KUKA KRL program: EPS_2_251806_MH46A_A_20260212042242.src

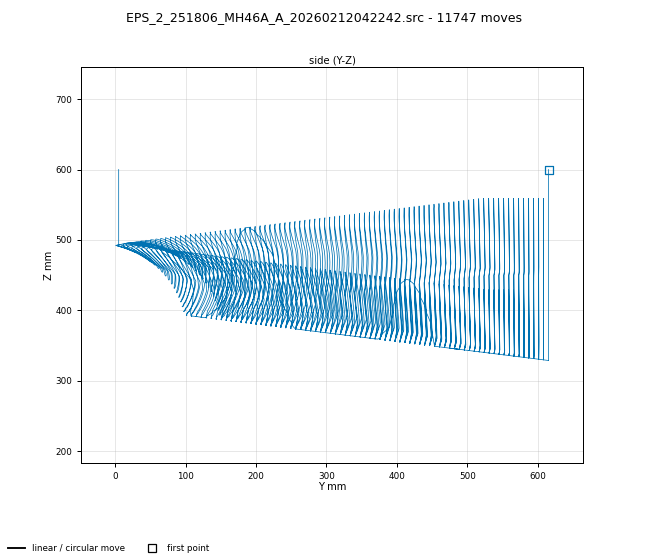
[picture p0: tool path of EPS_2_251806_MH46A_A_20260212042242.src, 11747 of 11749 moves have a stored position in this frame; points joined in program order, loops and branches not executed]
&ACCESS RVP
&REL 4
&COMMENT QRS 19112012
&PARAM EDITMASK = *
DEF PART()
EXT BAS (BAS_COMMAND :IN,REAL :IN )
INT I
BAS (#INITMOV,0 )

;KUKA QRS Post kuka4.cps  Date:22-06-2017 !

File_ID=3018

QRS_PRE_INIT()

;Init var - Until changes are made in qrs_pre_init
Outlet_Square_prg=0
Inlet_1_Square_prg=0
Inlet_2_Square_prg=0
Inlet_3_Square_prg=0
Inlet_4_Square_prg=0
Inlet_5_Square_prg=0

Outlet_1={X 0.000, Y 520.860, Z 458.500, B 0.000, E1 0.000 }
Inlet_1={X 0.000, Y 530.280, Z 328.500, B 0.000, E1 188.000 }
Outlet_1_type=201
Inlet_1_type=201
;QRS#1=Sidecore dimensions
;QRS#2=200-8" PVC SDR 35
;QRS#3=200-8" PVC SDR 35
;QRS#4=
;QRS#5=
;QRS#6=
;QRS#7=
;QRS#8=
;QRS#9=12-08 PSX
;QRS#10=12-08 PSX
;QRS#11=
;QRS#12=
;QRS#13=
;QRS#14=
;QRS#15=
;QRS#16=1220x127x838 2,75'
;QRS#17=EPS Height
;QRS#18=559
;QRS#19=*
;QRS#20= UPDATED VERSION 22-06-2017
;QRS#21=*
Outlet_Square=0100
Inlet_1_Square=0100
Inlet_2_Square=0
Inlet_3_Square=0
Inlet_4_Square=0
Inlet_5_Square=0
Mill_Square=1
Outlet_Square_Prg=204
Inlet_1_Square_prg=204

QRS_INIT()

$ADVANCE=5

; T1
PTP {E1 173.606,E2 173.606}
PTP {X 0,Y 615.511,A -85,B 0,C 180,E1 173.606,E2 173.606,E3 0,E4 0,E5 0,E6 0}
QRS_SPEED_INIT()
LIN {X 0,Y 615.511,Z 600,A -85,B 0,C 180,E1 173.606,E2 173.606,E3 0,E4 0,E5 0,E6 0} C_VEL
LIN {X 0,Y 615.511,Z 338.873,A -85,B 0,C 180,E1 173.606,E2 173.606} C_VEL
LIN {X 0,Y 615.511,Z 330.7,A -85,B 0,C 180,E1 173.606,E2 173.606} C_VEL
LIN {X 0,Y 615.495,Z 328.7,A -85,B 0,C 180,E1 173.42,E2 173.42} C_VEL
LIN {X 0,Y 615.496,Z 328.696,A -85,B 0,C 180,E1 170.801,E2 170.801} C_VEL
LIN {X 0,Y 615.477,Z 328.699,A -85,B 0,C 180,E1 168.139,E2 168.139} C_VEL
LIN {X 0,Y 615.495,Z 328.7,A -85,B 0,C 180,E1 165.451,E2 165.451} C_VEL
LIN {X 0,Y 615.495,Z 328.694,A -85,B 0,C 180,E1 162.729,E2 162.729} C_VEL
LIN {X 0,Y 615.493,Z 328.701,A -85,B 0,C 180,E1 159.967,E2 159.967} C_VEL
LIN {X 0,Y 615.487,Z 328.696,A -85,B 0,C 180,E1 157.155,E2 157.155} C_VEL
LIN {X 0,Y 615.499,Z 328.7,A -85,B 0,C 180,E1 154.284,E2 154.284} C_VEL
LIN {X 0,Y 615.478,Z 328.698,A -85,B 0,C 180,E1 151.552,E2 151.552} C_VEL
LIN {X 0,Y 615.492,Z 328.698,A -85,B 0,C 180,E1 148.914,E2 148.914} C_VEL
LIN {X 0,Y 615.498,Z 328.7,A -85,B 0,C 180,E1 146.465,E2 146.465} C_VEL
LIN {X 0,Y 615.494,Z 328.7,A -85,B 0,C 180,E1 144.166,E2 144.166} C_VEL
LIN {X 0,Y 615.491,Z 328.701,A -85,B 0,C 180,E1 141.931,E2 141.931} C_VEL
LIN {X 0,Y 615.491,Z 328.696,A -85,B 0,C 180,E1 139.393,E2 139.393} C_VEL
LIN {X 0,Y 615.482,Z 328.698,A -85,B 0,C 180,E1 136.754,E2 136.754} C_VEL
LIN {X 0,Y 615.491,Z 328.699,A -85,B 0,C 180,E1 133.997,E2 133.997} C_VEL
LIN {X 0,Y 615.493,Z 328.696,A -85,B 0,C 180,E1 131.094,E2 131.094} C_VEL
LIN {X 0,Y 615.484,Z 328.698,A -85,B 0,C 180,E1 128.905,E2 128.905} C_VEL
LIN {X 0,Y 615.49,Z 328.699,A -85,B 0,C 180,E1 126.425,E2 126.425} C_VEL
LIN {X 0,Y 615.496,Z 328.694,A -85,B 0,C 180,E1 123.534,E2 123.534} C_VEL
LIN {X 0,Y 615.487,Z 328.698,A -85,B 0,C 180,E1 120.92,E2 120.92} C_VEL
LIN {X 0,Y 615.498,Z 328.7,A -85,B 0,C 180,E1 118.451,E2 118.451} C_VEL
LIN {X 0,Y 615.499,Z 328.694,A -85,B 0,C 180,E1 115.57,E2 115.57} C_VEL
LIN {X 0,Y 615.492,Z 328.701,A -85,B 0,C 180,E1 112.845,E2 112.845} C_VEL
LIN {X 0,Y 615.482,Z 328.697,A -85,B 0,C 180,E1 110.033,E2 110.033} C_VEL
LIN {X 0,Y 615.495,Z 328.7,A -85,B 0,C 180,E1 107.271,E2 107.271} C_VEL
LIN {X 0,Y 615.484,Z 328.697,A -85,B 0,C 180,E1 104.55,E2 104.55} C_VEL
LIN {X 0,Y 615.49,Z 328.697,A -85,B 0,C 180,E1 101.861,E2 101.861} C_VEL
LIN {X 0,Y 615.495,Z 328.698,A -85,B 0,C 180,E1 99.199,E2 99.199} C_VEL
LIN {X 0,Y 615.479,Z 328.698,A -85,B 0,C 180,E1 96.557,E2 96.557} C_VEL
LIN {X 0,Y 615.488,Z 328.7,A -85,B 0,C 180,E1 93.601,E2 93.601} C_VEL
LIN {X 0,Y 615.482,Z 328.699,A -85,B 0,C 180,E1 93.478,E2 93.478} C_VEL
LIN {X 0,Y 615.482,Z 341.691,A -85,B 0,C 180,E1 93.151,E2 93.151} C_VEL
LIN {X 0,Y 615.495,Z 354.109,A -85,B 0,C 180,E1 92.7,E2 92.7} C_VEL
LIN {X 0,Y 615.492,Z 366.017,A -85,B 0,C 180,E1 92.127,E2 92.127} C_VEL
LIN {X 0,Y 615.495,Z 376.719,A -85,B 0,C 180,E1 91.473,E2 91.473} C_VEL
LIN {X 0,Y 615.498,Z 387.355,A -85,B 0,C 180,E1 90.655,E2 90.655} C_VEL
LIN {X 0,Y 615.499,Z 396.028,A -85,B 0,C 180,E1 89.837,E2 89.837} C_VEL
LIN {X 0,Y 615.496,Z 404.503,A -85,B 0,C 180,E1 88.856,E2 88.856} C_VEL
LIN {X 0,Y 615.496,Z 411.299,A -85,B 0,C 180,E1 87.874,E2 87.874} C_VEL
LIN {X 0,Y 615.497,Z 417.556,A -85,B 0,C 180,E1 86.728,E2 86.728} C_VEL
LIN {X 0,Y 615.495,Z 421.662,A -85,B 0,C 180,E1 85.744,E2 85.744} C_VEL
LIN {X 0,Y 615.495,Z 424.735,A -85,B 0,C 180,E1 84.759,E2 84.759} C_VEL
LIN {X 0,Y 615.499,Z 426.265,A -85,B 0,C 180,E1 84.102,E2 84.102} C_VEL
LIN {X 0,Y 615.496,Z 427.396,A -85,B 0,C 180,E1 83.42,E2 83.42} C_VEL
LIN {X 0,Y 615.497,Z 428.353,A -85,B 0,C 180,E1 82.125,E2 82.125} C_VEL
LIN {X 0,Y 615.494,Z 428.277,A -85,B 0,C 180,E1 81.464,E2 81.464} C_VEL
LIN {X 0,Y 615.497,Z 427.763,A -85,B 0,C 180,E1 80.802,E2 80.802} C_VEL
LIN {X 0,Y 615.499,Z 426.851,A -85,B 0,C 180,E1 80.138,E2 80.138} C_VEL
LIN {X 0,Y 615.494,Z 424.63,A -85,B 0,C 180,E1 79.112,E2 79.112} C_VEL
LIN {X 0,Y 615.494,Z 421.565,A -85,B 0,C 180,E1 78.14,E2 78.14} C_VEL
LIN {X 0,Y 615.498,Z 417.326,A -85,B 0,C 180,E1 77.135,E2 77.135} C_VEL
LIN {X 0,Y 615.497,Z 411.481,A -85,B 0,C 180,E1 76.066,E2 76.066} C_VEL
LIN {X 0,Y 615.496,Z 404.943,A -85,B 0,C 180,E1 75.113,E2 75.113} C_VEL
LIN {X 0,Y 615.499,Z 397.842,A -85,B 0,C 180,E1 74.266,E2 74.266} C_VEL
LIN {X 0,Y 615.497,Z 389.207,A -85,B 0,C 180,E1 73.414,E2 73.414} C_VEL
LIN {X 0,Y 615.498,Z 378.423,A -85,B 0,C 180,E1 72.559,E2 72.559} C_VEL
LIN {X 0,Y 615.482,Z 367.809,A -85,B 0,C 180,E1 71.881,E2 71.881} C_VEL
LIN {X 0,Y 615.493,Z 357.48,A -85,B 0,C 180,E1 71.355,E2 71.355} C_VEL
LIN {X 0,Y 615.48,Z 345.396,A -85,B 0,C 180,E1 70.879,E2 70.879} C_VEL
LIN {X 0,Y 615.491,Z 333.153,A -85,B 0,C 180,E1 70.533,E2 70.533} C_VEL
LIN {X 0,Y 615.492,Z 328.702,A -85,B 0,C 180,E1 70.424,E2 70.424} C_VEL
LIN {X 0,Y 615.483,Z 328.7,A -85,B 0,C 180,E1 67.656,E2 67.656} C_VEL
LIN {X 0,Y 615.479,Z 328.7,A -85,B 0,C 180,E1 65.008,E2 65.008} C_VEL
LIN {X 0,Y 615.476,Z 328.701,A -85,B 0,C 180,E1 62.823,E2 62.823} C_VEL
LIN {X 0,Y 615.482,Z 328.7,A -85,B 0,C 180,E1 60.207,E2 60.207} C_VEL
LIN {X 0,Y 615.494,Z 328.7,A -85,B 0,C 180,E1 57.543,E2 57.543} C_VEL
LIN {X 0,Y 615.484,Z 328.699,A -85,B 0,C 180,E1 55.185,E2 55.185} C_VEL
LIN {X 0,Y 615.488,Z 328.699,A -85,B 0,C 180,E1 52.759,E2 52.759} C_VEL
LIN {X 0,Y 615.482,Z 328.699,A -85,B 0,C 180,E1 49.912,E2 49.912} C_VEL
LIN {X 0,Y 615.499,Z 328.698,A -85,B 0,C 180,E1 47.649,E2 47.649} C_VEL
LIN {X 0,Y 615.486,Z 328.698,A -85,B 0,C 180,E1 44.932,E2 44.932} C_VEL
LIN {X 0,Y 615.485,Z 328.698,A -85,B 0,C 180,E1 42.081,E2 42.081} C_VEL
LIN {X 0,Y 615.497,Z 328.697,A -85,B 0,C 180,E1 39.75,E2 39.75} C_VEL
LIN {X 0,Y 615.492,Z 328.697,A -85,B 0,C 180,E1 36.938,E2 36.938} C_VEL
LIN {X 0,Y 615.497,Z 328.698,A -85,B 0,C 180,E1 34.703,E2 34.703} C_VEL
LIN {X 0,Y 615.482,Z 328.7,A -85,B 0,C 180,E1 32.331,E2 32.331} C_VEL
LIN {X 0,Y 615.496,Z 328.697,A -85,B 0,C 180,E1 29.797,E2 29.797} C_VEL
LIN {X 0,Y 615.499,Z 328.695,A -85,B 0,C 180,E1 27.048,E2 27.048} C_VEL
LIN {X 0,Y 615.492,Z 328.697,A -85,B 0,C 180,E1 24.272,E2 24.272} C_VEL
LIN {X 0,Y 615.495,Z 328.698,A -85,B 0,C 180,E1 21.432,E2 21.432} C_VEL
LIN {X 0,Y 615.495,Z 328.701,A -85,B 0,C 180,E1 18.608,E2 18.608} C_VEL
LIN {X 0,Y 615.489,Z 328.698,A -85,B 0,C 180,E1 15.905,E2 15.905} C_VEL
LIN {X 0,Y 615.496,Z 328.696,A -85,B 0,C 180,E1 13.201,E2 13.201} C_VEL
LIN {X 0,Y 615.495,Z 328.699,A -85,B 0,C 180,E1 10.527,E2 10.527} C_VEL
LIN {X 0,Y 615.485,Z 328.7,A -85,B 0,C 180,E1 7.876,E2 7.876} C_VEL
LIN {X 0,Y 615.491,Z 328.697,A -85,B 0,C 180,E1 5.241,E2 5.241} C_VEL
LIN {X 0,Y 615.496,Z 328.7,A -85,B 0,C 180,E1 2.618,E2 2.618} C_VEL
LIN {X 0,Y 615.484,Z 328.699,A -85,B 0,C 180,E1 0,E2 0} C_VEL
LIN {X 0,Y 615.49,Z 328.698,A -85,B 0,C 180,E1 -2.618,E2 -2.618} C_VEL
LIN {X 0,Y 615.497,Z 328.7,A -85,B 0,C 180,E1 -5.241,E2 -5.241} C_VEL
LIN {X 0,Y 615.479,Z 328.7,A -85,B 0,C 180,E1 -7.876,E2 -7.876} C_VEL
LIN {X 0,Y 615.487,Z 328.699,A -85,B 0,C 180,E1 -10.527,E2 -10.527} C_VEL
LIN {X 0,Y 615.496,Z 328.7,A -85,B 0,C 180,E1 -13.201,E2 -13.201} C_VEL
LIN {X 0,Y 615.477,Z 328.701,A -85,B 0,C 180,E1 -15.905,E2 -15.905} C_VEL
LIN {X 0,Y 615.479,Z 328.7,A -85,B 0,C 180,E1 -18.646,E2 -18.646} C_VEL
LIN {X 0,Y 615.485,Z 328.7,A -85,B 0,C 180,E1 -21.432,E2 -21.432} C_VEL
LIN {X 0,Y 615.489,Z 328.701,A -85,B 0,C 180,E1 -24.272,E2 -24.272} C_VEL
LIN {X 0,Y 615.493,Z 328.701,A -85,B 0,C 180,E1 -27.177,E2 -27.177} C_VEL
LIN {X 0,Y 615.499,Z 328.7,A -85,B 0,C 180,E1 -30.159,E2 -30.159} C_VEL
LIN {X 0,Y 615.485,Z 328.699,A -85,B 0,C 180,E1 -32.458,E2 -32.458} C_VEL
LIN {X 0,Y 615.491,Z 328.697,A -85,B 0,C 180,E1 -34.815,E2 -34.815} C_VEL
LIN {X 0,Y 615.495,Z 328.699,A -85,B 0,C 180,E1 -37.242,E2 -37.242} C_VEL
LIN {X 0,Y 615.498,Z 328.7,A -85,B 0,C 180,E1 -40.091,E2 -40.091} C_VEL
LIN {X 0,Y 615.492,Z 328.7,A -85,B 0,C 180,E1 -43.049,E2 -43.049} C_VEL
LIN {X 0,Y 615.49,Z 328.7,A -85,B 0,C 180,E1 -46.002,E2 -46.002} C_VEL
LIN {X 0,Y 615.496,Z 328.698,A -85,B 0,C 180,E1 -48.905,E2 -48.905} C_VEL
LIN {X 0,Y 615.497,Z 328.701,A -85,B 0,C 180,E1 -51.097,E2 -51.097} C_VEL
LIN {X 0,Y 615.492,Z 328.697,A -85,B 0,C 180,E1 -53.576,E2 -53.576} C_VEL
LIN {X 0,Y 615.489,Z 328.805,A -85,B 0,C 180,E1 -54.611,E2 -54.611} C_VEL
LIN {X 0,Y 615.491,Z 341.278,A -85,B 0,C 180,E1 -57.155,E2 -57.155} C_VEL
LIN {X 0,Y 615.495,Z 354.171,A -85,B 0,C 180,E1 -59.841,E2 -59.841} C_VEL
LIN {X 0,Y 615.495,Z 366.88,A -85,B 0,C 180,E1 -62.455,E2 -62.455} C_VEL
LIN {X 0,Y 615.478,Z 379.58,A -85,B 0,C 180,E1 -65.008,E2 -65.008} C_VEL
LIN {X 0,Y 615.484,Z 394.081,A -85,B 0,C 180,E1 -67.864,E2 -67.864} C_VEL
LIN {X 0,Y 615.485,Z 408.57,A -85,B 0,C 180,E1 -70.663,E2 -70.663} C_VEL
LIN {X 0,Y 615.496,Z 423.857,A -85,B 0,C 180,E1 -73.567,E2 -73.567} C_VEL
LIN {X 0,Y 615.493,Z 439.318,A -85,B 0,C 180,E1 -76.463,E2 -76.463} C_VEL
LIN {X 0,Y 615.49,Z 449.367,A -85,B 0,C 180,E1 -78.328,E2 -78.328} C_VEL
LIN {X 0,Y 615.478,Z 464.088,A -85,B 0,C 180,E1 -78.599,E2 -78.599} C_VEL
LIN {X 0,Y 615.481,Z 476.501,A -85,B 0,C 180,E1 -78.96,E2 -78.96} C_VEL
LIN {X 0,Y 615.481,Z 489.034,A -85,B 0,C 180,E1 -79.473,E2 -79.473} C_VEL
LIN {X 0,Y 615.491,Z 499.989,A -85,B 0,C 180,E1 -80.055,E2 -80.055} C_VEL
LIN {X 0,Y 615.499,Z 511.174,A -85,B 0,C 180,E1 -80.802,E2 -80.802} C_VEL
LIN {X 0,Y 615.498,Z 521.05,A -85,B 0,C 180,E1 -81.629,E2 -81.629} C_VEL
LIN {X 0,Y 615.498,Z 530.61,A -85,B 0,C 180,E1 -82.62,E2 -82.62} C_VEL
LIN {X 0,Y 615.496,Z 538.206,A -85,B 0,C 180,E1 -83.609,E2 -83.609} C_VEL
LIN {X 0,Y 615.498,Z 545.207,A -85,B 0,C 180,E1 -84.759,E2 -84.759} C_VEL
LIN {X 0,Y 615.493,Z 549.854,A -85,B 0,C 180,E1 -85.744,E2 -85.744} C_VEL
LIN {X 0,Y 615.495,Z 553.4,A -85,B 0,C 180,E1 -86.728,E2 -86.728} C_VEL
LIN {X 0,Y 615.497,Z 555.234,A -85,B 0,C 180,E1 -87.383,E2 -87.383} C_VEL
LIN {X 0,Y 615.499,Z 556.608,A -85,B 0,C 180,E1 -88.037,E2 -88.037} C_VEL
LIN {X 0,Y 615.496,Z 558.174,A -85,B 0,C 180,E1 -89.346,E2 -89.346} C_VEL
LIN {X 0,Y 615.494,Z 558.389,A -85,B 0,C 180,E1 -90,E2 -90} C_VEL
LIN {X 0,Y 615.496,Z 557.579,A -85,B 0,C 180,E1 -91.309,E2 -91.309} C_VEL
LIN {X 0,Y 615.499,Z 556.607,A -85,B 0,C 180,E1 -91.964,E2 -91.964} C_VEL
LIN {X 0,Y 615.497,Z 555.232,A -85,B 0,C 180,E1 -92.618,E2 -92.618} C_VEL
LIN {X 0,Y 615.496,Z 552.348,A -85,B 0,C 180,E1 -93.601,E2 -93.601} C_VEL
LIN {X 0,Y 615.498,Z 548.439,A -85,B 0,C 180,E1 -94.585,E2 -94.585} C_VEL
LIN {X 0,Y 615.499,Z 543.402,A -85,B 0,C 180,E1 -95.57,E2 -95.57} C_VEL
LIN {X 0,Y 615.497,Z 536.869,A -85,B 0,C 180,E1 -96.583,E2 -96.583} C_VEL
LIN {X 0,Y 615.497,Z 529.129,A -85,B 0,C 180,E1 -97.546,E2 -97.546} C_VEL
LIN {X 0,Y 615.498,Z 521.04,A -85,B 0,C 180,E1 -98.372,E2 -98.372} C_VEL
LIN {X 0,Y 615.499,Z 511.161,A -85,B 0,C 180,E1 -99.199,E2 -99.199} C_VEL
LIN {X 0,Y 615.491,Z 499.973,A -85,B 0,C 180,E1 -99.946,E2 -99.946} C_VEL
LIN {X 0,Y 615.481,Z 489.013,A -85,B 0,C 180,E1 -100.527,E2 -100.527} C_VEL
LIN {X 0,Y 615.484,Z 476.479,A -85,B 0,C 180,E1 -101.04,E2 -101.04} C_VEL
LIN {X 0,Y 615.478,Z 464.046,A -85,B 0,C 180,E1 -101.402,E2 -101.402} C_VEL
LIN {X 0,Y 615.49,Z 449.249,A -85,B 0,C 180,E1 -101.694,E2 -101.694} C_VEL
LIN {X 0,Y 615.483,Z 433.893,A -85,B 0,C 180,E1 -104.55,E2 -104.55} C_VEL
LIN {X 0,Y 615.478,Z 419.426,A -85,B 0,C 180,E1 -107.271,E2 -107.271} C_VEL
LIN {X 0,Y 615.479,Z 404.947,A -85,B 0,C 180,E1 -110.034,E2 -110.034} C_VEL
LIN {X 0,Y 615.492,Z 390.453,A -85,B 0,C 180,E1 -112.845,E2 -112.845} C_VEL
LIN {X 0,Y 615.492,Z 375.947,A -85,B 0,C 180,E1 -115.716,E2 -115.716} C_VEL
LIN {X 0,Y 615.491,Z 362.442,A -85,B 0,C 180,E1 -118.451,E2 -118.451} C_VEL
LIN {X 0,Y 615.485,Z 349.75,A -85,B 0,C 180,E1 -121.085,E2 -121.085} C_VEL
LIN {X 0,Y 615.495,Z 337.872,A -85,B 0,C 180,E1 -123.535,E2 -123.535} C_VEL
LIN {X 0,Y 615.488,Z 328.696,A -85,B 0,C 180,E1 -125.466,E2 -125.466} C_VEL
LIN {X 0,Y 615.483,Z 328.7,A -85,B 0,C 180,E1 -128.069,E2 -128.069} C_VEL
LIN {X 0,Y 615.492,Z 328.7,A -85,B 0,C 180,E1 -130.607,E2 -130.607} C_VEL
LIN {X 0,Y 615.497,Z 328.694,A -85,B 0,C 180,E1 -133.244,E2 -133.244} C_VEL
LIN {X 0,Y 615.484,Z 328.701,A -85,B 0,C 180,E1 -136.004,E2 -136.004} C_VEL
LIN {X 0,Y 615.483,Z 328.697,A -85,B 0,C 180,E1 -138.907,E2 -138.907} C_VEL
LIN {X 0,Y 615.493,Z 328.695,A -85,B 0,C 180,E1 -141.096,E2 -141.096} C_VEL
LIN {X 0,Y 615.478,Z 328.699,A -85,B 0,C 180,E1 -143.574,E2 -143.574} C_VEL
LIN {X 0,Y 615.489,Z 328.698,A -85,B 0,C 180,E1 -145.978,E2 -145.978} C_VEL
LIN {X 0,Y 615.495,Z 328.698,A -85,B 0,C 180,E1 -148.315,E2 -148.315} C_VEL
LIN {X 0,Y 615.49,Z 328.699,A -85,B 0,C 180,E1 -150.594,E2 -150.594} C_VEL
LIN {X 0,Y 615.497,Z 328.7,A -85,B 0,C 180,E1 -152.954,E2 -152.954} C_VEL
LIN {X 0,Y 615.492,Z 328.695,A -85,B 0,C 180,E1 -155.728,E2 -155.728} C_VEL
LIN {X 0,Y 615.498,Z 328.7,A -85,B 0,C 180,E1 -158.569,E2 -158.569} C_VEL
LIN {X 0,Y 615.477,Z 328.699,A -85,B 0,C 180,E1 -161.4,E2 -161.4} C_VEL
LIN {X 0,Y 615.494,Z 328.699,A -85,B 0,C 180,E1 -164.095,E2 -164.095} C_VEL
LIN {X 0,Y 615.494,Z 328.696,A -85,B 0,C 180,E1 -166.799,E2 -166.799} C_VEL
LIN {X 0,Y 615.486,Z 328.698,A -85,B 0,C 180,E1 -169.473,E2 -169.473} C_VEL
LIN {X 0,Y 615.492,Z 328.7,A -85,B 0,C 180,E1 -172.125,E2 -172.125} C_VEL
LIN {X 0,Y 615.488,Z 328.696,A -85,B 0,C 180,E1 -174.759,E2 -174.759} C_VEL
LIN {X 0,Y 615.488,Z 328.698,A -85,B 0,C 180,E1 -177.382,E2 -177.382} C_VEL
LIN {X 0,Y 615.492,Z 328.7,A -85,B 0,C 180,E1 -180,E2 -180} C_VEL
LIN {X 0,Y 615.489,Z 328.696,A -85,B 0,C 180,E1 -182.618,E2 -182.618} C_VEL
LIN {X 0,Y 615.487,Z 328.698,A -85,B 0,C 180,E1 -185.241,E2 -185.241} C_VEL
LIN {X 0,Y 615.495,Z 328.7,A -85,B 0,C 180,E1 -186.58,E2 -186.58} C_VEL
LIN {X 0,Y 614.816,Z 328.843,A -85,B 0,C 180,E1 -187.126,E2 -187.126} C_VEL
LIN {X 0,Y 611.983,Z 329.256,A -85,B 0,C 180,E1 -188.012,E2 -188.012} C_VEL
LIN {X 0,Y 609.593,Z 329.565,A -85,B 0,C 180,E1 -188.724,E2 -188.724} C_VEL
LIN {X 0,Y 608.558,Z 329.683,A -85,B 0,C 180,E1 -189.274,E2 -189.274} C_VEL
LIN {X 0,Y 608.468,Z 329.693,A -85,B 0,C 180,E1 -189.46,E2 -189.46} C_VEL
LIN {X 0,Y 608.456,Z 329.696,A -85,B 0,C 180,E1 -192,E2 -192} C_VEL
LIN {X 0,Y 608.483,Z 329.692,A -85,B 0,C 180,E1 -194.721,E2 -194.721} C_VEL
LIN {X 0,Y 608.462,Z 329.694,A -85,B 0,C 180,E1 -197.477,E2 -197.477} C_VEL
LIN {X 0,Y 608.462,Z 329.695,A -85,B 0,C 180,E1 -200.274,E2 -200.274} C_VEL
LIN {X 0,Y 608.452,Z 329.696,A -85,B 0,C 180,E1 -203.124,E2 -203.124} C_VEL
LIN {X 0,Y 608.481,Z 329.695,A -85,B 0,C 180,E1 -205.722,E2 -205.722} C_VEL
LIN {X 0,Y 608.447,Z 329.696,A -85,B 0,C 180,E1 -208.267,E2 -208.267} C_VEL
LIN {X 0,Y 608.48,Z 329.692,A -85,B 0,C 180,E1 -210.545,E2 -210.545} C_VEL
LIN {X 0,Y 608.466,Z 329.693,A -85,B 0,C 180,E1 -212.879,E2 -212.879} C_VEL
LIN {X 0,Y 608.448,Z 329.695,A -85,B 0,C 180,E1 -215.278,E2 -215.278} C_VEL
LIN {X 0,Y 608.473,Z 329.694,A -85,B 0,C 180,E1 -218.24,E2 -218.24} C_VEL
LIN {X 0,Y 608.458,Z 329.697,A -85,B 0,C 180,E1 -220.329,E2 -220.329} C_VEL
LIN {X 0,Y 608.471,Z 329.693,A -85,B 0,C 180,E1 -223.308,E2 -223.308} C_VEL
LIN {X 0,Y 608.477,Z 329.693,A -85,B 0,C 180,E1 -226.131,E2 -226.131} C_VEL
LIN {X 0,Y 608.462,Z 329.694,A -85,B 0,C 180,E1 -228.823,E2 -228.823} C_VEL
LIN {X 0,Y 608.465,Z 329.694,A -85,B 0,C 180,E1 -231.761,E2 -231.761} C_VEL
LIN {X 0,Y 608.451,Z 329.696,A -85,B 0,C 180,E1 -233.955,E2 -233.955} C_VEL
LIN {X 0,Y 608.473,Z 329.693,A -85,B 0,C 180,E1 -236.329,E2 -236.329} C_VEL
LIN {X 0,Y 608.453,Z 329.695,A -85,B 0,C 180,E1 -238.732,E2 -238.732} C_VEL
LIN {X 0,Y 608.479,Z 329.693,A -85,B 0,C 180,E1 -241.38,E2 -241.38} C_VEL
LIN {X 0,Y 608.48,Z 329.691,A -85,B 0,C 180,E1 -244.279,E2 -244.279} C_VEL
LIN {X 0,Y 608.457,Z 329.695,A -85,B 0,C 180,E1 -246.876,E2 -246.876} C_VEL
LIN {X 0,Y 608.463,Z 329.694,A -85,B 0,C 180,E1 -249.725,E2 -249.725} C_VEL
LIN {X 0,Y 608.461,Z 329.695,A -85,B 0,C 180,E1 -252.523,E2 -252.523} C_VEL
LIN {X 0,Y 608.475,Z 329.693,A -85,B 0,C 180,E1 -255.279,E2 -255.279} C_VEL
LIN {X 0,Y 608.466,Z 329.693,A -85,B 0,C 180,E1 -258,E2 -258} C_VEL
LIN {X 0,Y 608.479,Z 329.695,A -85,B 0,C 180,E1 -260.694,E2 -260.694} C_VEL
LIN {X 0,Y 608.465,Z 329.693,A -85,B 0,C 180,E1 -263.384,E2 -263.384} C_VEL
LIN {X 0,Y 608.471,Z 329.695,A -85,B 0,C 180,E1 -266.357,E2 -266.357} C_VEL
LIN {X 0,Y 608.47,Z 329.695,A -85,B 0,C 180,E1 -266.399,E2 -266.399} C_VEL
LIN {X 0,Y 608.537,Z 344.673,A -85,B 0,C 180,E1 -266.813,E2 -266.813} C_VEL
LIN {X 0,Y 608.528,Z 356.437,A -85,B 0,C 180,E1 -267.269,E2 -267.269} C_VEL
LIN {X 0,Y 608.501,Z 367.879,A -85,B 0,C 180,E1 -267.848,E2 -267.848} C_VEL
LIN {X 0,Y 608.484,Z 379.387,A -85,B 0,C 180,E1 -268.593,E2 -268.593} C_VEL
LIN {X 0,Y 608.492,Z 388.706,A -85,B 0,C 180,E1 -269.338,E2 -269.338} C_VEL
LIN {X 0,Y 608.469,Z 397.258,A -85,B 0,C 180,E1 -270.165,E2 -270.165} C_VEL
LIN {X 0,Y 608.452,Z 405.583,A -85,B 0,C 180,E1 -271.158,E2 -271.158} C_VEL
LIN {X 0,Y 608.453,Z 412.309,A -85,B 0,C 180,E1 -272.151,E2 -272.151} C_VEL
LIN {X 0,Y 608.432,Z 418.509,A -85,B 0,C 180,E1 -273.31,E2 -273.31} C_VEL
LIN {X 0,Y 608.441,Z 422.549,A -85,B 0,C 180,E1 -274.305,E2 -274.305} C_VEL
LIN {X 0,Y 608.438,Z 425.557,A -85,B 0,C 180,E1 -275.302,E2 -275.302} C_VEL
LIN {X 0,Y 608.435,Z 427.044,A -85,B 0,C 180,E1 -275.967,E2 -275.967} C_VEL
LIN {X 0,Y 608.449,Z 428.079,A -85,B 0,C 180,E1 -276.632,E2 -276.632} C_VEL
LIN {X 0,Y 608.422,Z 428.988,A -85,B 0,C 180,E1 -277.967,E2 -277.967} C_VEL
LIN {X 0,Y 608.418,Z 428.833,A -85,B 0,C 180,E1 -278.636,E2 -278.636} C_VEL
LIN {X 0,Y 608.434,Z 427.29,A -85,B 0,C 180,E1 -279.977,E2 -279.977} C_VEL
LIN {X 0,Y 608.423,Z 425.177,A -85,B 0,C 180,E1 -280.931,E2 -280.931} C_VEL
LIN {X 0,Y 608.444,Z 421.748,A -85,B 0,C 180,E1 -282,E2 -282} C_VEL
LIN {X 0,Y 608.431,Z 417.356,A -85,B 0,C 180,E1 -283.017,E2 -283.017} C_VEL
LIN {X 0,Y 608.456,Z 411.712,A -85,B 0,C 180,E1 -284.037,E2 -284.037} C_VEL
LIN {X 0,Y 608.446,Z 404.61,A -85,B 0,C 180,E1 -285.063,E2 -285.063} C_VEL
LIN {X 0,Y 608.462,Z 395.624,A -85,B 0,C 180,E1 -286.093,E2 -286.093} C_VEL
LIN {X 0,Y 608.485,Z 386.353,A -85,B 0,C 180,E1 -286.955,E2 -286.955} C_VEL
LIN {X 0,Y 608.489,Z 376,A -85,B 0,C 180,E1 -287.735,E2 -287.735} C_VEL
LIN {X 0,Y 608.493,Z 364.686,A -85,B 0,C 180,E1 -288.416,E2 -288.416} C_VEL
LIN {X 0,Y 608.505,Z 352.29,A -85,B 0,C 180,E1 -288.999,E2 -288.999} C_VEL
LIN {X 0,Y 608.536,Z 339.565,A -85,B 0,C 180,E1 -289.436,E2 -289.436} C_VEL
LIN {X 0,Y 608.459,Z 329.697,A -85,B 0,C 180,E1 -289.702,E2 -289.702} C_VEL
LIN {X 0,Y 608.463,Z 329.696,A -85,B 0,C 180,E1 -292.476,E2 -292.476} C_VEL
LIN {X 0,Y 608.453,Z 329.696,A -85,B 0,C 180,E1 -295.3,E2 -295.3} C_VEL
LIN {X 0,Y 608.444,Z 329.699,A -85,B 0,C 180,E1 -297.518,E2 -297.518} C_VEL
LIN {X 0,Y 608.463,Z 329.694,A -85,B 0,C 180,E1 -299.97,E2 -299.97} C_VEL
LIN {X 0,Y 608.46,Z 329.695,A -85,B 0,C 180,E1 -302.879,E2 -302.879} C_VEL
LIN {X 0,Y 608.446,Z 329.697,A -85,B 0,C 180,E1 -305.277,E2 -305.277} C_VEL
LIN {X 0,Y 608.467,Z 329.694,A -85,B 0,C 180,E1 -307.746,E2 -307.746} C_VEL
LIN {X 0,Y 608.452,Z 329.697,A -85,B 0,C 180,E1 -310.328,E2 -310.328} C_VEL
LIN {X 0,Y 608.48,Z 329.693,A -85,B 0,C 180,E1 -313.309,E2 -313.309} C_VEL
LIN {X 0,Y 608.47,Z 329.694,A -85,B 0,C 180,E1 -316.13,E2 -316.13} C_VEL
LIN {X 0,Y 608.459,Z 329.695,A -85,B 0,C 180,E1 -318.823,E2 -318.823} C_VEL
LIN {X 0,Y 608.474,Z 329.695,A -85,B 0,C 180,E1 -321.412,E2 -321.412} C_VEL
LIN {X 0,Y 608.48,Z 329.692,A -85,B 0,C 180,E1 -323.949,E2 -323.949} C_VEL
LIN {X 0,Y 608.472,Z 329.695,A -85,B 0,C 180,E1 -326.329,E2 -326.329} C_VEL
LIN {X 0,Y 608.479,Z 329.692,A -85,B 0,C 180,E1 -328.727,E2 -328.727} C_VEL
LIN {X 0,Y 608.478,Z 329.694,A -85,B 0,C 180,E1 -331.378,E2 -331.378} C_VEL
LIN {X 0,Y 608.452,Z 329.696,A -85,B 0,C 180,E1 -333.964,E2 -333.964} C_VEL
LIN {X 0,Y 608.474,Z 329.694,A -85,B 0,C 180,E1 -336.155,E2 -336.155} C_VEL
LIN {X 0,Y 608.46,Z 329.695,A -85,B 0,C 180,E1 -339.018,E2 -339.018} C_VEL
LIN {X 0,Y 608.454,Z 329.695,A -85,B 0,C 180,E1 -341.828,E2 -341.828} C_VEL
LIN {X 0,Y 608.477,Z 329.693,A -85,B 0,C 180,E1 -344.594,E2 -344.594} C_VEL
LIN {X 0,Y 608.485,Z 329.694,A -85,B 0,C 180,E1 -347.323,E2 -347.323} C_VEL
LIN {X 0,Y 608.455,Z 329.696,A -85,B 0,C 180,E1 -350.022,E2 -350.022} C_VEL
LIN {X 0,Y 608.464,Z 329.694,A -85,B 0,C 180,E1 -352.7,E2 -352.7} C_VEL
LIN {X 0,Y 608.465,Z 329.696,A -85,B 0,C 180,E1 -355.362,E2 -355.362} C_VEL
LIN {X 0,Y 608.452,Z 329.696,A -85,B 0,C 180,E1 -358.014,E2 -358.014} C_VEL
LIN {X 0,Y 608.483,Z 329.692,A -85,B 0,C 180,E1 -360.662,E2 -360.662} C_VEL
LIN {X 0,Y 608.484,Z 329.694,A -85,B 0,C 180,E1 -363.311,E2 -363.311} C_VEL
LIN {X 0,Y 608.456,Z 329.695,A -85,B 0,C 180,E1 -365.967,E2 -365.967} C_VEL
LIN {X 0,Y 608.457,Z 329.695,A -85,B 0,C 180,E1 -368.636,E2 -368.636} C_VEL
LIN {X 0,Y 608.478,Z 329.694,A -85,B 0,C 180,E1 -371.324,E2 -371.324} C_VEL
LIN {X 0,Y 608.465,Z 329.695,A -85,B 0,C 180,E1 -374.037,E2 -374.037} C_VEL
LIN {X 0,Y 608.472,Z 329.693,A -85,B 0,C 180,E1 -376.783,E2 -376.783} C_VEL
LIN {X 0,Y 608.455,Z 329.696,A -85,B 0,C 180,E1 -379.57,E2 -379.57} C_VEL
LIN {X 0,Y 608.455,Z 329.696,A -85,B 0,C 180,E1 -382.477,E2 -382.477} C_VEL
LIN {X 0,Y 608.457,Z 329.695,A -85,B 0,C 180,E1 -384.571,E2 -384.571} C_VEL
LIN {X 0,Y 608.486,Z 329.694,A -85,B 0,C 180,E1 -387.21,E2 -387.21} C_VEL
LIN {X 0,Y 608.472,Z 329.694,A -85,B 0,C 180,E1 -389.973,E2 -389.973} C_VEL
LIN {X 0,Y 608.46,Z 329.695,A -85,B 0,C 180,E1 -392.523,E2 -392.523} C_VEL
LIN {X 0,Y 608.445,Z 329.698,A -85,B 0,C 180,E1 -395.278,E2 -395.278} C_VEL
LIN {X 0,Y 608.478,Z 329.693,A -85,B 0,C 180,E1 -397.746,E2 -397.746} C_VEL
LIN {X 0,Y 608.48,Z 329.693,A -85,B 0,C 180,E1 -400.333,E2 -400.333} C_VEL
LIN {X 0,Y 608.481,Z 329.693,A -85,B 0,C 180,E1 -403.311,E2 -403.311} C_VEL
LIN {X 0,Y 608.475,Z 329.695,A -85,B 0,C 180,E1 -406.132,E2 -406.132} C_VEL
LIN {X 0,Y 608.464,Z 329.695,A -85,B 0,C 180,E1 -408.825,E2 -408.825} C_VEL
LIN {X 0,Y 608.477,Z 329.693,A -85,B 0,C 180,E1 -411.413,E2 -411.413} C_VEL
LIN {X 0,Y 608.486,Z 329.693,A -85,B 0,C 180,E1 -414.319,E2 -414.319} C_VEL
LIN {X 0,Y 608.492,Z 329.891,A -85,B 0,C 180,E1 -414.473,E2 -414.473} C_VEL
LIN {X 0,Y 608.546,Z 340.78,A -85,B 0,C 180,E1 -416.732,E2 -416.732} C_VEL
LIN {X 0,Y 608.584,Z 352.391,A -85,B 0,C 180,E1 -419.085,E2 -419.085} C_VEL
LIN {X 0,Y 608.557,Z 365.066,A -85,B 0,C 180,E1 -421.739,E2 -421.739} C_VEL
LIN {X 0,Y 608.532,Z 378.505,A -85,B 0,C 180,E1 -424.484,E2 -424.484} C_VEL
LIN {X 0,Y 608.53,Z 392.306,A -85,B 0,C 180,E1 -427.239,E2 -427.239} C_VEL
LIN {X 0,Y 608.482,Z 406.831,A -85,B 0,C 180,E1 -430.079,E2 -430.079} C_VEL
LIN {X 0,Y 608.469,Z 421.358,A -85,B 0,C 180,E1 -432.871,E2 -432.871} C_VEL
LIN {X 0,Y 608.459,Z 435.885,A -85,B 0,C 180,E1 -435.621,E2 -435.621} C_VEL
LIN {X 0,Y 608.473,Z 449.882,A -85,B 0,C 180,E1 -438.202,E2 -438.202} C_VEL
LIN {X 0,Y 608.54,Z 463.289,A -85,B 0,C 180,E1 -438.446,E2 -438.446} C_VEL
LIN {X 0,Y 608.522,Z 475.912,A -85,B 0,C 180,E1 -438.808,E2 -438.808} C_VEL
LIN {X 0,Y 608.515,Z 487.605,A -85,B 0,C 180,E1 -439.276,E2 -439.276} C_VEL
LIN {X 0,Y 608.491,Z 498.764,A -85,B 0,C 180,E1 -439.856,E2 -439.856} C_VEL
LIN {X 0,Y 608.504,Z 510.259,A -85,B 0,C 180,E1 -440.611,E2 -440.611} C_VEL
LIN {X 0,Y 608.472,Z 519.542,A -85,B 0,C 180,E1 -441.365,E2 -441.365} C_VEL
LIN {X 0,Y 608.455,Z 527.993,A -85,B 0,C 180,E1 -442.2,E2 -442.2} C_VEL
LIN {X 0,Y 608.462,Z 536.239,A -85,B 0,C 180,E1 -443.201,E2 -443.201} C_VEL
LIN {X 0,Y 608.437,Z 542.879,A -85,B 0,C 180,E1 -444.2,E2 -444.2} C_VEL
LIN {X 0,Y 608.432,Z 548.952,A -85,B 0,C 180,E1 -445.363,E2 -445.363} C_VEL
LIN {X 0,Y 608.449,Z 552.898,A -85,B 0,C 180,E1 -446.358,E2 -446.358} C_VEL
LIN {X 0,Y 608.425,Z 555.81,A -85,B 0,C 180,E1 -447.352,E2 -447.352} C_VEL
LIN {X 0,Y 608.444,Z 557.202,A -85,B 0,C 180,E1 -448.015,E2 -448.015} C_VEL
LIN {X 0,Y 608.438,Z 558.784,A -85,B 0,C 180,E1 -449.339,E2 -449.339} C_VEL
LIN {X 0,Y 608.434,Z 559,A -85,B 0,C 180,E1 -450,E2 -450} C_VEL
LIN {X 0,Y 608.448,Z 558.183,A -85,B 0,C 180,E1 -451.324,E2 -451.324} C_VEL
LIN {X 0,Y 608.444,Z 557.201,A -85,B 0,C 180,E1 -451.986,E2 -451.986} C_VEL
LIN {X 0,Y 608.425,Z 555.808,A -85,B 0,C 180,E1 -452.649,E2 -452.649} C_VEL
LIN {X 0,Y 608.449,Z 552.895,A -85,B 0,C 180,E1 -453.643,E2 -453.643} C_VEL
LIN {X 0,Y 608.432,Z 548.948,A -85,B 0,C 180,E1 -454.638,E2 -454.638} C_VEL
LIN {X 0,Y 608.437,Z 542.874,A -85,B 0,C 180,E1 -455.801,E2 -455.801} C_VEL
LIN {X 0,Y 608.462,Z 536.231,A -85,B 0,C 180,E1 -456.8,E2 -456.8} C_VEL
LIN {X 0,Y 608.456,Z 527.985,A -85,B 0,C 180,E1 -457.801,E2 -457.801} C_VEL
LIN {X 0,Y 608.472,Z 519.531,A -85,B 0,C 180,E1 -458.636,E2 -458.636} C_VEL
LIN {X 0,Y 608.481,Z 509.084,A -85,B 0,C 180,E1 -459.474,E2 -459.474} C_VEL
LIN {X 0,Y 608.491,Z 498.747,A -85,B 0,C 180,E1 -460.145,E2 -460.145} C_VEL
LIN {X 0,Y 608.518,Z 487.257,A -85,B 0,C 180,E1 -460.74,E2 -460.74} C_VEL
LIN {X 0,Y 608.529,Z 474.881,A -85,B 0,C 180,E1 -461.225,E2 -461.225} C_VEL
LIN {X 0,Y 608.542,Z 461.418,A -85,B 0,C 180,E1 -461.597,E2 -461.597} C_VEL
LIN {X 0,Y 608.448,Z 449.612,A -85,B 0,C 180,E1 -461.81,E2 -461.81} C_VEL
LIN {X 0,Y 608.46,Z 435.879,A -85,B 0,C 180,E1 -464.38,E2 -464.38} C_VEL
LIN {X 0,Y 608.471,Z 421.353,A -85,B 0,C 180,E1 -467.13,E2 -467.13} C_VEL
LIN {X 0,Y 608.482,Z 406.826,A -85,B 0,C 180,E1 -469.922,E2 -469.922} C_VEL
LIN {X 0,Y 608.512,Z 392.301,A -85,B 0,C 180,E1 -472.762,E2 -472.762} C_VEL
LIN {X 0,Y 608.532,Z 378.502,A -85,B 0,C 180,E1 -475.517,E2 -475.517} C_VEL
LIN {X 0,Y 608.557,Z 365.061,A -85,B 0,C 180,E1 -478.262,E2 -478.262} C_VEL
LIN {X 0,Y 608.584,Z 352.394,A -85,B 0,C 180,E1 -480.915,E2 -480.915} C_VEL
LIN {X 0,Y 608.567,Z 338.438,A -85,B 0,C 180,E1 -483.748,E2 -483.748} C_VEL
LIN {X 0,Y 608.472,Z 329.693,A -85,B 0,C 180,E1 -485.606,E2 -485.606} C_VEL
LIN {X 0,Y 608.465,Z 329.696,A -85,B 0,C 180,E1 -488.24,E2 -488.24} C_VEL
LIN {X 0,Y 608.467,Z 329.694,A -85,B 0,C 180,E1 -491.343,E2 -491.343} C_VEL
LIN {X 0,Y 608.465,Z 329.694,A -85,B 0,C 180,E1 -494.264,E2 -494.264} C_VEL
LIN {X 0,Y 608.448,Z 329.697,A -85,B 0,C 180,E1 -497.04,E2 -497.04} C_VEL
LIN {X 0,Y 608.457,Z 329.696,A -85,B 0,C 180,E1 -499.697,E2 -499.697} C_VEL
LIN {X 0,Y 608.477,Z 329.692,A -85,B 0,C 180,E1 -502.254,E2 -502.254} C_VEL
LIN {X 0,Y 608.457,Z 329.698,A -85,B 0,C 180,E1 -505.094,E2 -505.094} C_VEL
LIN {X 0,Y 608.471,Z 329.692,A -85,B 0,C 180,E1 -507.906,E2 -507.906} C_VEL
LIN {X 0,Y 608.47,Z 329.693,A -85,B 0,C 180,E1 -510.221,E2 -510.221} C_VEL
LIN {X 0,Y 608.484,Z 329.693,A -85,B 0,C 180,E1 -512.793,E2 -512.793} C_VEL
LIN {X 0,Y 608.487,Z 329.691,A -85,B 0,C 180,E1 -515.847,E2 -515.847} C_VEL
LIN {X 0,Y 608.48,Z 329.692,A -85,B 0,C 180,E1 -518.309,E2 -518.309} C_VEL
LIN {X 0,Y 608.468,Z 329.693,A -85,B 0,C 180,E1 -521.286,E2 -521.286} C_VEL
LIN {X 0,Y 608.467,Z 329.694,A -85,B 0,C 180,E1 -523.906,E2 -523.906} C_VEL
LIN {X 0,Y 608.47,Z 329.694,A -85,B 0,C 180,E1 -526.644,E2 -526.644} C_VEL
LIN {X 0,Y 608.462,Z 329.694,A -85,B 0,C 180,E1 -529.35,E2 -529.35} C_VEL
LIN {X 0,Y 608.483,Z 329.694,A -85,B 0,C 180,E1 -532.033,E2 -532.033} C_VEL
LIN {X 0,Y 608.468,Z 329.693,A -85,B 0,C 180,E1 -534.698,E2 -534.698} C_VEL
LIN {X 0,Y 608.479,Z 329.692,A -85,B 0,C 180,E1 -537.352,E2 -537.352} C_VEL
LIN {X 0,Y 608.483,Z 329.693,A -85,B 0,C 180,E1 -540,E2 -540} C_VEL
LIN {X 0,Y 608.48,Z 329.691,A -85,B 0,C 180,E1 -542.648,E2 -542.648} C_VEL
LIN {X 0,Y 608.466,Z 329.695,A -85,B 0,C 180,E1 -545.302,E2 -545.302} C_VEL
LIN {X 0,Y 608.48,Z 329.693,A -85,B 0,C 180,E1 -547.967,E2 -547.967} C_VEL
LIN {X 0,Y 608.468,Z 329.693,A -85,B 0,C 180,E1 -549.46,E2 -549.46} C_VEL
LIN {X 0,Y 607.785,Z 329.781,A -85,B 0,C 180,E1 -550.013,E2 -550.013} C_VEL
LIN {X 0,Y 604.925,Z 330.138,A -85,B 0,C 180,E1 -550.91,E2 -550.91} C_VEL
LIN {X 0,Y 602.52,Z 330.437,A -85,B 0,C 180,E1 -551.631,E2 -551.631} C_VEL
LIN {X 0,Y 601.491,Z 330.565,A -85,B 0,C 180,E1 -552.188,E2 -552.188} C_VEL
LIN {X 0,Y 601.408,Z 330.573,A -85,B 0,C 180,E1 -552.376,E2 -552.376} C_VEL
LIN {X 0,Y 601.437,Z 330.569,A -85,B 0,C 180,E1 -554.897,E2 -554.897} C_VEL
LIN {X 0,Y 601.441,Z 330.569,A -85,B 0,C 180,E1 -556.986,E2 -556.986} C_VEL
LIN {X 0,Y 601.409,Z 330.573,A -85,B 0,C 180,E1 -559.81,E2 -559.81} C_VEL
LIN {X 0,Y 601.418,Z 330.571,A -85,B 0,C 180,E1 -562.683,E2 -562.683} C_VEL
LIN {X 0,Y 601.41,Z 330.573,A -85,B 0,C 180,E1 -564.879,E2 -564.879} C_VEL
LIN {X 0,Y 601.423,Z 330.57,A -85,B 0,C 180,E1 -567.363,E2 -567.363} C_VEL
LIN {X 0,Y 601.435,Z 330.572,A -85,B 0,C 180,E1 -570.164,E2 -570.164} C_VEL
LIN {X 0,Y 601.431,Z 330.57,A -85,B 0,C 180,E1 -572.716,E2 -572.716} C_VEL
LIN {X 0,Y 601.406,Z 330.573,A -85,B 0,C 180,E1 -575.113,E2 -575.113} C_VEL
LIN {X 0,Y 601.439,Z 330.569,A -85,B 0,C 180,E1 -577.419,E2 -577.419} C_VEL
LIN {X 0,Y 601.418,Z 330.572,A -85,B 0,C 180,E1 -579.995,E2 -579.995} C_VEL
LIN {X 0,Y 601.415,Z 330.573,A -85,B 0,C 180,E1 -582.671,E2 -582.671} C_VEL
LIN {X 0,Y 601.434,Z 330.57,A -85,B 0,C 180,E1 -585.482,E2 -585.482} C_VEL
LIN {X 0,Y 601.432,Z 330.57,A -85,B 0,C 180,E1 -588.407,E2 -588.407} C_VEL
LIN {X 0,Y 601.411,Z 330.572,A -85,B 0,C 180,E1 -590.873,E2 -590.873} C_VEL
LIN {X 0,Y 601.401,Z 330.574,A -85,B 0,C 180,E1 -593.416,E2 -593.416} C_VEL
LIN {X 0,Y 601.44,Z 330.571,A -85,B 0,C 180,E1 -596.064,E2 -596.064} C_VEL
LIN {X 0,Y 601.427,Z 330.571,A -85,B 0,C 180,E1 -598.545,E2 -598.545} C_VEL
LIN {X 0,Y 601.438,Z 330.57,A -85,B 0,C 180,E1 -601.373,E2 -601.373} C_VEL
LIN {X 0,Y 601.42,Z 330.572,A -85,B 0,C 180,E1 -604.132,E2 -604.132} C_VEL
LIN {X 0,Y 601.425,Z 330.57,A -85,B 0,C 180,E1 -606.589,E2 -606.589} C_VEL
LIN {X 0,Y 601.435,Z 330.572,A -85,B 0,C 180,E1 -609.478,E2 -609.478} C_VEL
LIN {X 0,Y 601.405,Z 330.573,A -85,B 0,C 180,E1 -612.311,E2 -612.311} C_VEL
LIN {X 0,Y 601.419,Z 330.571,A -85,B 0,C 180,E1 -614.408,E2 -614.408} C_VEL
LIN {X 0,Y 601.42,Z 330.573,A -85,B 0,C 180,E1 -617.171,E2 -617.171} C_VEL
LIN {X 0,Y 601.445,Z 330.568,A -85,B 0,C 180,E1 -619.905,E2 -619.905} C_VEL
LIN {X 0,Y 601.449,Z 330.568,A -85,B 0,C 180,E1 -622.614,E2 -622.614} C_VEL
LIN {X 0,Y 601.42,Z 330.573,A -85,B 0,C 180,E1 -625.307,E2 -625.307} C_VEL
LIN {X 0,Y 601.456,Z 330.758,A -85,B 0,C 180,E1 -626.294,E2 -626.294} C_VEL
LIN {X 0,Y 601.573,Z 343.736,A -85,B 0,C 180,E1 -626.651,E2 -626.651} C_VEL
LIN {X 0,Y 601.535,Z 356.698,A -85,B 0,C 180,E1 -627.153,E2 -627.153} C_VEL
LIN {X 0,Y 601.513,Z 368.062,A -85,B 0,C 180,E1 -627.74,E2 -627.74} C_VEL
LIN {X 0,Y 601.471,Z 379.541,A -85,B 0,C 180,E1 -628.493,E2 -628.493} C_VEL
LIN {X 0,Y 601.432,Z 389.788,A -85,B 0,C 180,E1 -629.33,E2 -629.33} C_VEL
LIN {X 0,Y 601.414,Z 399.587,A -85,B 0,C 180,E1 -630.334,E2 -630.334} C_VEL
LIN {X 0,Y 601.384,Z 407.507,A -85,B 0,C 180,E1 -631.339,E2 -631.339} C_VEL
LIN {X 0,Y 601.365,Z 413.865,A -85,B 0,C 180,E1 -632.344,E2 -632.344} C_VEL
LIN {X 0,Y 601.351,Z 418.937,A -85,B 0,C 180,E1 -633.35,E2 -633.35} C_VEL
LIN {X 0,Y 601.355,Z 422.885,A -85,B 0,C 180,E1 -634.356,E2 -634.356} C_VEL
LIN {X 0,Y 601.349,Z 425.806,A -85,B 0,C 180,E1 -635.364,E2 -635.364} C_VEL
LIN {X 0,Y 601.349,Z 428.041,A -85,B 0,C 180,E1 -636.583,E2 -636.583} C_VEL
LIN {X 0,Y 601.322,Z 428.791,A -85,B 0,C 180,E1 -637.386,E2 -637.386} C_VEL
LIN {X 0,Y 601.333,Z 428.999,A -85,B 0,C 180,E1 -638.062,E2 -638.062} C_VEL
LIN {X 0,Y 601.336,Z 428.147,A -85,B 0,C 180,E1 -639.417,E2 -639.417} C_VEL
LIN {X 0,Y 601.33,Z 427.132,A -85,B 0,C 180,E1 -640.096,E2 -640.096} C_VEL
LIN {X 0,Y 601.336,Z 425.175,A -85,B 0,C 180,E1 -640.966,E2 -640.966} C_VEL
LIN {X 0,Y 601.366,Z 421.393,A -85,B 0,C 180,E1 -642.143,E2 -642.143} C_VEL
LIN {X 0,Y 601.348,Z 416.889,A -85,B 0,C 180,E1 -643.173,E2 -643.173} C_VEL
LIN {X 0,Y 601.383,Z 411.126,A -85,B 0,C 180,E1 -644.206,E2 -644.206} C_VEL
LIN {X 0,Y 601.38,Z 403.833,A -85,B 0,C 180,E1 -645.244,E2 -645.244} C_VEL
LIN {X 0,Y 601.407,Z 394.672,A -85,B 0,C 180,E1 -646.287,E2 -646.287} C_VEL
LIN {X 0,Y 601.447,Z 385.17,A -85,B 0,C 180,E1 -647.16,E2 -647.16} C_VEL
LIN {X 0,Y 601.485,Z 374.505,A -85,B 0,C 180,E1 -647.949,E2 -647.949} C_VEL
LIN {X 0,Y 601.525,Z 363.252,A -85,B 0,C 180,E1 -648.616,E2 -648.616} C_VEL
LIN {X 0,Y 601.546,Z 352.015,A -85,B 0,C 180,E1 -649.138,E2 -649.138} C_VEL
LIN {X 0,Y 601.567,Z 339.146,A -85,B 0,C 180,E1 -649.581,E2 -649.581} C_VEL
LIN {X 0,Y 601.426,Z 330.572,A -85,B 0,C 180,E1 -649.808,E2 -649.808} C_VEL
LIN {X 0,Y 601.416,Z 330.574,A -85,B 0,C 180,E1 -652.682,E2 -652.682} C_VEL
LIN {X 0,Y 601.402,Z 330.574,A -85,B 0,C 180,E1 -654.878,E2 -654.878} C_VEL
LIN {X 0,Y 601.41,Z 330.574,A -85,B 0,C 180,E1 -657.36,E2 -657.36} C_VEL
LIN {X 0,Y 601.43,Z 330.571,A -85,B 0,C 180,E1 -660.148,E2 -660.148} C_VEL
LIN {X 0,Y 601.427,Z 330.572,A -85,B 0,C 180,E1 -662.715,E2 -662.715} C_VEL
LIN {X 0,Y 601.4,Z 330.574,A -85,B 0,C 180,E1 -665.112,E2 -665.112} C_VEL
LIN {X 0,Y 601.436,Z 330.572,A -85,B 0,C 180,E1 -667.418,E2 -667.418} C_VEL
LIN {X 0,Y 601.403,Z 330.574,A -85,B 0,C 180,E1 -669.995,E2 -669.995} C_VEL
LIN {X 0,Y 601.416,Z 330.573,A -85,B 0,C 180,E1 -672.669,E2 -672.669} C_VEL
LIN {X 0,Y 601.426,Z 330.574,A -85,B 0,C 180,E1 -675.481,E2 -675.481} C_VEL
LIN {X 0,Y 601.428,Z 330.573,A -85,B 0,C 180,E1 -678.406,E2 -678.406} C_VEL
LIN {X 0,Y 601.439,Z 330.569,A -85,B 0,C 180,E1 -680.875,E2 -680.875} C_VEL
LIN {X 0,Y 601.446,Z 330.569,A -85,B 0,C 180,E1 -683.733,E2 -683.733} C_VEL
LIN {X 0,Y 601.438,Z 330.57,A -85,B 0,C 180,E1 -686.063,E2 -686.063} C_VEL
LIN {X 0,Y 601.443,Z 330.57,A -85,B 0,C 180,E1 -688.541,E2 -688.541} C_VEL
LIN {X 0,Y 601.438,Z 330.571,A -85,B 0,C 180,E1 -691.373,E2 -691.373} C_VEL
LIN {X 0,Y 601.41,Z 330.574,A -85,B 0,C 180,E1 -693.636,E2 -693.636} C_VEL
LIN {X 0,Y 601.427,Z 330.571,A -85,B 0,C 180,E1 -696.59,E2 -696.59} C_VEL
LIN {X 0,Y 601.435,Z 330.571,A -85,B 0,C 180,E1 -699.478,E2 -699.478} C_VEL
LIN {X 0,Y 601.404,Z 330.575,A -85,B 0,C 180,E1 -702.312,E2 -702.312} C_VEL
LIN {X 0,Y 601.421,Z 330.574,A -85,B 0,C 180,E1 -704.409,E2 -704.409} C_VEL
LIN {X 0,Y 601.43,Z 330.571,A -85,B 0,C 180,E1 -707.172,E2 -707.172} C_VEL
LIN {X 0,Y 601.434,Z 330.57,A -85,B 0,C 180,E1 -709.905,E2 -709.905} C_VEL
LIN {X 0,Y 601.441,Z 330.569,A -85,B 0,C 180,E1 -712.615,E2 -712.615} C_VEL
LIN {X 0,Y 601.432,Z 330.572,A -85,B 0,C 180,E1 -715.308,E2 -715.308} C_VEL
LIN {X 0,Y 601.423,Z 330.572,A -85,B 0,C 180,E1 -717.991,E2 -717.991} C_VEL
LIN {X 0,Y 601.454,Z 330.567,A -85,B 0,C 180,E1 -720.669,E2 -720.669} C_VEL
LIN {X 0,Y 601.435,Z 330.572,A -85,B 0,C 180,E1 -723.349,E2 -723.349} C_VEL
LIN {X 0,Y 601.41,Z 330.573,A -85,B 0,C 180,E1 -726.037,E2 -726.037} C_VEL
LIN {X 0,Y 601.437,Z 330.569,A -85,B 0,C 180,E1 -728.738,E2 -728.738} C_VEL
LIN {X 0,Y 601.434,Z 330.571,A -85,B 0,C 180,E1 -731.458,E2 -731.458} C_VEL
LIN {X 0,Y 601.416,Z 330.574,A -85,B 0,C 180,E1 -734.205,E2 -734.205} C_VEL
LIN {X 0,Y 601.431,Z 330.571,A -85,B 0,C 180,E1 -736.986,E2 -736.986} C_VEL
LIN {X 0,Y 601.407,Z 330.573,A -85,B 0,C 180,E1 -739.809,E2 -739.809} C_VEL
LIN {X 0,Y 601.409,Z 330.573,A -85,B 0,C 180,E1 -742.683,E2 -742.683} C_VEL
LIN {X 0,Y 601.404,Z 330.574,A -85,B 0,C 180,E1 -744.878,E2 -744.878} C_VEL
LIN {X 0,Y 601.422,Z 330.572,A -85,B 0,C 180,E1 -747.867,E2 -747.867} C_VEL
LIN {X 0,Y 601.447,Z 330.571,A -85,B 0,C 180,E1 -750.163,E2 -750.163} C_VEL
LIN {X 0,Y 601.422,Z 330.571,A -85,B 0,C 180,E1 -752.716,E2 -752.716} C_VEL
LIN {X 0,Y 601.413,Z 330.575,A -85,B 0,C 180,E1 -755.115,E2 -755.115} C_VEL
LIN {X 0,Y 601.437,Z 330.57,A -85,B 0,C 180,E1 -757.419,E2 -757.419} C_VEL
LIN {X 0,Y 601.416,Z 330.574,A -85,B 0,C 180,E1 -759.995,E2 -759.995} C_VEL
LIN {X 0,Y 601.412,Z 330.573,A -85,B 0,C 180,E1 -762.67,E2 -762.67} C_VEL
LIN {X 0,Y 601.424,Z 330.571,A -85,B 0,C 180,E1 -765.483,E2 -765.483} C_VEL
LIN {X 0,Y 601.43,Z 330.571,A -85,B 0,C 180,E1 -768.406,E2 -768.406} C_VEL
LIN {X 0,Y 601.441,Z 330.57,A -85,B 0,C 180,E1 -770.876,E2 -770.876} C_VEL
LIN {X 0,Y 601.446,Z 330.569,A -85,B 0,C 180,E1 -773.734,E2 -773.734} C_VEL
LIN {X 0,Y 601.465,Z 330.628,A -85,B 0,C 180,E1 -774.251,E2 -774.251} C_VEL
LIN {X 0,Y 601.647,Z 336.403,A -85,B 0,C 180,E1 -775.491,E2 -775.491} C_VEL
LIN {X 0,Y 601.621,Z 351.103,A -85,B 0,C 180,E1 -778.514,E2 -778.514} C_VEL
LIN {X 0,Y 601.661,Z 361.435,A -85,B 0,C 180,E1 -780.62,E2 -780.62} C_VEL
LIN {X 0,Y 601.614,Z 374.146,A -85,B 0,C 180,E1 -783.273,E2 -783.273} C_VEL
LIN {X 0,Y 601.545,Z 388.672,A -85,B 0,C 180,E1 -786.23,E2 -786.23} C_VEL
LIN {X 0,Y 601.49,Z 401.383,A -85,B 0,C 180,E1 -788.764,E2 -788.764} C_VEL
LIN {X 0,Y 601.468,Z 414.772,A -85,B 0,C 180,E1 -791.389,E2 -791.389} C_VEL
LIN {X 0,Y 601.428,Z 428.621,A -85,B 0,C 180,E1 -794.062,E2 -794.062} C_VEL
LIN {X 0,Y 601.402,Z 443.148,A -85,B 0,C 180,E1 -796.828,E2 -796.828} C_VEL
LIN {X 0,Y 601.412,Z 449.882,A -85,B 0,C 180,E1 -798.061,E2 -798.061} C_VEL
LIN {X 0,Y 601.577,Z 462.375,A -85,B 0,C 180,E1 -798.289,E2 -798.289} C_VEL
LIN {X 0,Y 601.555,Z 475.414,A -85,B 0,C 180,E1 -798.661,E2 -798.661} C_VEL
LIN {X 0,Y 601.528,Z 487.604,A -85,B 0,C 180,E1 -799.15,E2 -799.15} C_VEL
LIN {X 0,Y 601.469,Z 498.765,A -85,B 0,C 180,E1 -799.736,E2 -799.736} C_VEL
LIN {X 0,Y 601.462,Z 510.26,A -85,B 0,C 180,E1 -800.5,E2 -800.5} C_VEL
LIN {X 0,Y 601.436,Z 519.542,A -85,B 0,C 180,E1 -801.263,E2 -801.263} C_VEL
LIN {X 0,Y 601.4,Z 527.994,A -85,B 0,C 180,E1 -802.108,E2 -802.108} C_VEL
LIN {X 0,Y 601.381,Z 536.239,A -85,B 0,C 180,E1 -803.121,E2 -803.121} C_VEL
LIN {X 0,Y 601.372,Z 542.88,A -85,B 0,C 180,E1 -804.131,E2 -804.131} C_VEL
LIN {X 0,Y 601.336,Z 548.952,A -85,B 0,C 180,E1 -805.308,E2 -805.308} C_VEL
LIN {X 0,Y 601.367,Z 552.898,A -85,B 0,C 180,E1 -806.315,E2 -806.315} C_VEL
LIN {X 0,Y 601.325,Z 555.81,A -85,B 0,C 180,E1 -807.321,E2 -807.321} C_VEL
LIN {X 0,Y 601.343,Z 557.202,A -85,B 0,C 180,E1 -807.991,E2 -807.991} C_VEL
LIN {X 0,Y 601.339,Z 558.784,A -85,B 0,C 180,E1 -809.331,E2 -809.331} C_VEL
LIN {X 0,Y 601.335,Z 559,A -85,B 0,C 180,E1 -810,E2 -810} C_VEL
LIN {X 0,Y 601.348,Z 558.184,A -85,B 0,C 180,E1 -811.34,E2 -811.34} C_VEL
LIN {X 0,Y 601.343,Z 557.201,A -85,B 0,C 180,E1 -812.01,E2 -812.01} C_VEL
LIN {X 0,Y 601.325,Z 555.808,A -85,B 0,C 180,E1 -812.68,E2 -812.68} C_VEL
LIN {X 0,Y 601.367,Z 552.894,A -85,B 0,C 180,E1 -813.686,E2 -813.686} C_VEL
LIN {X 0,Y 601.336,Z 548.948,A -85,B 0,C 180,E1 -814.693,E2 -814.693} C_VEL
LIN {X 0,Y 601.372,Z 542.874,A -85,B 0,C 180,E1 -815.87,E2 -815.87} C_VEL
LIN {X 0,Y 601.382,Z 536.232,A -85,B 0,C 180,E1 -816.88,E2 -816.88} C_VEL
LIN {X 0,Y 601.4,Z 527.985,A -85,B 0,C 180,E1 -817.893,E2 -817.893} C_VEL
LIN {X 0,Y 601.436,Z 519.531,A -85,B 0,C 180,E1 -818.738,E2 -818.738} C_VEL
LIN {X 0,Y 601.451,Z 509.085,A -85,B 0,C 180,E1 -819.586,E2 -819.586} C_VEL
LIN {X 0,Y 601.469,Z 498.749,A -85,B 0,C 180,E1 -820.265,E2 -820.265} C_VEL
LIN {X 0,Y 601.537,Z 486.598,A -85,B 0,C 180,E1 -820.896,E2 -820.896} C_VEL
LIN {X 0,Y 601.562,Z 474.205,A -85,B 0,C 180,E1 -821.379,E2 -821.379} C_VEL
LIN {X 0,Y 601.592,Z 461.417,A -85,B 0,C 180,E1 -821.733,E2 -821.733} C_VEL
LIN {X 0,Y 601.414,Z 449.612,A -85,B 0,C 180,E1 -821.95,E2 -821.95} C_VEL
LIN {X 0,Y 601.42,Z 435.879,A -85,B 0,C 180,E1 -824.552,E2 -824.552} C_VEL
LIN {X 0,Y 601.444,Z 421.353,A -85,B 0,C 180,E1 -827.336,E2 -827.336} C_VEL
LIN {X 0,Y 601.477,Z 406.826,A -85,B 0,C 180,E1 -830.164,E2 -830.164} C_VEL
LIN {X 0,Y 601.55,Z 394.115,A -85,B 0,C 180,E1 -832.678,E2 -832.678} C_VEL
LIN {X 0,Y 601.566,Z 381.404,A -85,B 0,C 180,E1 -835.241,E2 -835.241} C_VEL
LIN {X 0,Y 601.628,Z 368.693,A -85,B 0,C 180,E1 -837.857,E2 -837.857} C_VEL
LIN {X 0,Y 601.677,Z 355.875,A -85,B 0,C 180,E1 -840.538,E2 -840.538} C_VEL
LIN {X 0,Y 601.607,Z 340.631,A -85,B 0,C 180,E1 -843.633,E2 -843.633} C_VEL
LIN {X 0,Y 601.65,Z 332.298,A -85,B 0,C 180,E1 -845.4,E2 -845.4} C_VEL
LIN {X 0,Y 601.442,Z 330.571,A -85,B 0,C 180,E1 -845.796,E2 -845.796} C_VEL
LIN {X 0,Y 601.416,Z 330.573,A -85,B 0,C 180,E1 -848.469,E2 -848.469} C_VEL
LIN {X 0,Y 601.418,Z 330.572,A -85,B 0,C 180,E1 -850.875,E2 -850.875} C_VEL
LIN {X 0,Y 601.455,Z 330.567,A -85,B 0,C 180,E1 -853.584,E2 -853.584} C_VEL
LIN {X 0,Y 601.433,Z 330.57,A -85,B 0,C 180,E1 -856.428,E2 -856.428} C_VEL
LIN {X 0,Y 601.421,Z 330.573,A -85,B 0,C 180,E1 -859.427,E2 -859.427} C_VEL
LIN {X 0,Y 601.43,Z 330.573,A -85,B 0,C 180,E1 -861.733,E2 -861.733} C_VEL
LIN {X 0,Y 601.392,Z 330.576,A -85,B 0,C 180,E1 -864.246,E2 -864.246} C_VEL
LIN {X 0,Y 601.421,Z 330.571,A -85,B 0,C 180,E1 -866.686,E2 -866.686} C_VEL
LIN {X 0,Y 601.437,Z 330.569,A -85,B 0,C 180,E1 -869.059,E2 -869.059} C_VEL
LIN {X 0,Y 601.43,Z 330.57,A -85,B 0,C 180,E1 -871.373,E2 -871.373} C_VEL
LIN {X 0,Y 601.402,Z 330.573,A -85,B 0,C 180,E1 -873.636,E2 -873.636} C_VEL
LIN {X 0,Y 601.428,Z 330.571,A -85,B 0,C 180,E1 -876.59,E2 -876.59} C_VEL
LIN {X 0,Y 601.428,Z 330.571,A -85,B 0,C 180,E1 -879.478,E2 -879.478} C_VEL
LIN {X 0,Y 601.401,Z 330.574,A -85,B 0,C 180,E1 -882.312,E2 -882.312} C_VEL
LIN {X 0,Y 601.422,Z 330.572,A -85,B 0,C 180,E1 -884.409,E2 -884.409} C_VEL
LIN {X 0,Y 601.422,Z 330.571,A -85,B 0,C 180,E1 -887.172,E2 -887.172} C_VEL
LIN {X 0,Y 601.431,Z 330.572,A -85,B 0,C 180,E1 -889.905,E2 -889.905} C_VEL
LIN {X 0,Y 601.447,Z 330.567,A -85,B 0,C 180,E1 -892.615,E2 -892.615} C_VEL
LIN {X 0,Y 601.433,Z 330.572,A -85,B 0,C 180,E1 -895.308,E2 -895.308} C_VEL
LIN {X 0,Y 601.422,Z 330.571,A -85,B 0,C 180,E1 -897.991,E2 -897.991} C_VEL
LIN {X 0,Y 601.457,Z 330.567,A -85,B 0,C 180,E1 -900.67,E2 -900.67} C_VEL
LIN {X 0,Y 601.435,Z 330.572,A -85,B 0,C 180,E1 -903.35,E2 -903.35} C_VEL
LIN {X 0,Y 601.411,Z 330.572,A -85,B 0,C 180,E1 -906.037,E2 -906.037} C_VEL
LIN {X 0,Y 601.444,Z 330.57,A -85,B 0,C 180,E1 -908.738,E2 -908.738} C_VEL
LIN {X 0,Y 601.441,Z 330.569,A -85,B 0,C 180,E1 -911.458,E2 -911.458} C_VEL
LIN {X 0,Y 601.408,Z 330.573,A -85,B 0,C 180,E1 -912.376,E2 -912.376} C_VEL
LIN {X 0,Y 600.746,Z 330.655,A -85,B 0,C 180,E1 -912.936,E2 -912.936} C_VEL
LIN {X 0,Y 597.9,Z 331.009,A -85,B 0,C 180,E1 -913.843,E2 -913.843} C_VEL
LIN {X 0,Y 595.491,Z 331.312,A -85,B 0,C 180,E1 -914.574,E2 -914.574} C_VEL
LIN {X 0,Y 594.453,Z 331.439,A -85,B 0,C 180,E1 -915.137,E2 -915.137} C_VEL
LIN {X 0,Y 594.367,Z 331.449,A -85,B 0,C 180,E1 -915.328,E2 -915.328} C_VEL
LIN {X 0,Y 594.385,Z 331.45,A -85,B 0,C 180,E1 -917.904,E2 -917.904} C_VEL
LIN {X 0,Y 594.376,Z 331.449,A -85,B 0,C 180,E1 -920.914,E2 -920.914} C_VEL
LIN {X 0,Y 594.395,Z 331.447,A -85,B 0,C 180,E1 -923.704,E2 -923.704} C_VEL
LIN {X 0,Y 594.392,Z 331.449,A -85,B 0,C 180,E1 -926.7,E2 -926.7} C_VEL
LIN {X 0,Y 594.381,Z 331.45,A -85,B 0,C 180,E1 -928.999,E2 -928.999} C_VEL
LIN {X 0,Y 594.384,Z 331.448,A -85,B 0,C 180,E1 -931.643,E2 -931.643} C_VEL
LIN {X 0,Y 594.391,Z 331.449,A -85,B 0,C 180,E1 -934.58,E2 -934.58} C_VEL
LIN {X 0,Y 594.395,Z 331.446,A -85,B 0,C 180,E1 -937.608,E2 -937.608} C_VEL
LIN {X 0,Y 594.378,Z 331.449,A -85,B 0,C 180,E1 -940.567,E2 -940.567} C_VEL
LIN {X 0,Y 594.372,Z 331.449,A -85,B 0,C 180,E1 -943.3,E2 -943.3} C_VEL
LIN {X 0,Y 594.39,Z 331.447,A -85,B 0,C 180,E1 -946.159,E2 -946.159} C_VEL
LIN {X 0,Y 594.384,Z 331.45,A -85,B 0,C 180,E1 -949.178,E2 -949.178} C_VEL
LIN {X 0,Y 594.387,Z 331.447,A -85,B 0,C 180,E1 -952.059,E2 -952.059} C_VEL
LIN {X 0,Y 594.356,Z 331.452,A -85,B 0,C 180,E1 -954.677,E2 -954.677} C_VEL
LIN {X 0,Y 594.387,Z 331.45,A -85,B 0,C 180,E1 -957.088,E2 -957.088} C_VEL
LIN {X 0,Y 594.376,Z 331.449,A -85,B 0,C 180,E1 -959.675,E2 -959.675} C_VEL
LIN {X 0,Y 594.382,Z 331.449,A -85,B 0,C 180,E1 -962.539,E2 -962.539} C_VEL
LIN {X 0,Y 594.384,Z 331.449,A -85,B 0,C 180,E1 -964.807,E2 -964.807} C_VEL
LIN {X 0,Y 594.373,Z 331.451,A -85,B 0,C 180,E1 -967.264,E2 -967.264} C_VEL
LIN {X 0,Y 594.378,Z 331.448,A -85,B 0,C 180,E1 -969.946,E2 -969.946} C_VEL
LIN {X 0,Y 594.397,Z 331.449,A -85,B 0,C 180,E1 -972.806,E2 -972.806} C_VEL
LIN {X 0,Y 594.396,Z 331.446,A -85,B 0,C 180,E1 -975.826,E2 -975.826} C_VEL
LIN {X 0,Y 594.387,Z 331.45,A -85,B 0,C 180,E1 -978.404,E2 -978.404} C_VEL
LIN {X 0,Y 594.388,Z 331.447,A -85,B 0,C 180,E1 -981.157,E2 -981.157} C_VEL
LIN {X 0,Y 594.37,Z 331.451,A -85,B 0,C 180,E1 -983.891,E2 -983.891} C_VEL
LIN {X 0,Y 594.389,Z 331.45,A -85,B 0,C 180,E1 -986.165,E2 -986.165} C_VEL
LIN {X 0,Y 594.609,Z 337.876,A -85,B 0,C 180,E1 -986.336,E2 -986.336} C_VEL
LIN {X 0,Y 594.577,Z 351.028,A -85,B 0,C 180,E1 -986.781,E2 -986.781} C_VEL
LIN {X 0,Y 594.514,Z 362.151,A -85,B 0,C 180,E1 -987.289,E2 -987.289} C_VEL
LIN {X 0,Y 594.448,Z 373.677,A -85,B 0,C 180,E1 -987.967,E2 -987.967} C_VEL
LIN {X 0,Y 594.435,Z 385.078,A -85,B 0,C 180,E1 -988.814,E2 -988.814} C_VEL
LIN {X 0,Y 594.363,Z 394.258,A -85,B 0,C 180,E1 -989.661,E2 -989.661} C_VEL
LIN {X 0,Y 594.341,Z 403.175,A -85,B 0,C 180,E1 -990.677,E2 -990.677} C_VEL
LIN {X 0,Y 594.283,Z 410.391,A -85,B 0,C 180,E1 -991.694,E2 -991.694} C_VEL
LIN {X 0,Y 594.253,Z 416.184,A -85,B 0,C 180,E1 -992.711,E2 -992.711} C_VEL
LIN {X 0,Y 594.288,Z 420.756,A -85,B 0,C 180,E1 -993.729,E2 -993.729} C_VEL
LIN {X 0,Y 594.23,Z 424.249,A -85,B 0,C 180,E1 -994.748,E2 -994.748} C_VEL
LIN {X 0,Y 594.263,Z 426.023,A -85,B 0,C 180,E1 -995.428,E2 -995.428} C_VEL
LIN {X 0,Y 594.274,Z 428.302,A -85,B 0,C 180,E1 -996.791,E2 -996.791} C_VEL
LIN {X 0,Y 594.247,Z 428.857,A -85,B 0,C 180,E1 -997.475,E2 -997.475} C_VEL
LIN {X 0,Y 594.229,Z 428.98,A -85,B 0,C 180,E1 -998.159,E2 -998.159} C_VEL
LIN {X 0,Y 594.256,Z 428.035,A -85,B 0,C 180,E1 -999.53,E2 -999.53} C_VEL
LIN {X 0,Y 594.231,Z 426.958,A -85,B 0,C 180,E1 -1000.218,E2 -1000.218} C_VEL
LIN {X 0,Y 594.251,Z 425.17,A -85,B 0,C 180,E1 -1001.002,E2 -1001.002} C_VEL
LIN {X 0,Y 594.258,Z 421.033,A -85,B 0,C 180,E1 -1002.291,E2 -1002.291} C_VEL
LIN {X 0,Y 594.274,Z 416.419,A -85,B 0,C 180,E1 -1003.333,E2 -1003.333} C_VEL
LIN {X 0,Y 594.306,Z 410.505,A -85,B 0,C 180,E1 -1004.379,E2 -1004.379} C_VEL
LIN {X 0,Y 594.34,Z 403.044,A -85,B 0,C 180,E1 -1005.429,E2 -1005.429} C_VEL
LIN {X 0,Y 594.364,Z 393.714,A -85,B 0,C 180,E1 -1006.486,E2 -1006.486} C_VEL
LIN {X 0,Y 594.431,Z 383.932,A -85,B 0,C 180,E1 -1007.369,E2 -1007.369} C_VEL
LIN {X 0,Y 594.466,Z 372.998,A -85,B 0,C 180,E1 -1008.168,E2 -1008.168} C_VEL
LIN {X 0,Y 594.554,Z 362.308,A -85,B 0,C 180,E1 -1008.792,E2 -1008.792} C_VEL
LIN {X 0,Y 594.566,Z 350.566,A -85,B 0,C 180,E1 -1009.327,E2 -1009.327} C_VEL
LIN {X 0,Y 594.625,Z 337.949,A -85,B 0,C 180,E1 -1009.752,E2 -1009.752} C_VEL
LIN {X 0,Y 594.552,Z 332.32,A -85,B 0,C 180,E1 -1009.898,E2 -1009.898} C_VEL
LIN {X 0,Y 594.391,Z 331.448,A -85,B 0,C 180,E1 -1009.94,E2 -1009.94} C_VEL
LIN {X 0,Y 594.367,Z 331.45,A -85,B 0,C 180,E1 -1012.967,E2 -1012.967} C_VEL
LIN {X 0,Y 594.378,Z 331.449,A -85,B 0,C 180,E1 -1015.192,E2 -1015.192} C_VEL
LIN {X 0,Y 594.371,Z 331.452,A -85,B 0,C 180,E1 -1017.523,E2 -1017.523} C_VEL
LIN {X 0,Y 594.387,Z 331.449,A -85,B 0,C 180,E1 -1020.327,E2 -1020.327} C_VEL
LIN {X 0,Y 594.382,Z 331.449,A -85,B 0,C 180,E1 -1022.949,E2 -1022.949} C_VEL
LIN {X 0,Y 594.353,Z 331.454,A -85,B 0,C 180,E1 -1025.408,E2 -1025.408} C_VEL
LIN {X 0,Y 594.386,Z 331.448,A -85,B 0,C 180,E1 -1027.94,E2 -1027.94} C_VEL
LIN {X 0,Y 594.381,Z 331.449,A -85,B 0,C 180,E1 -1030.822,E2 -1030.822} C_VEL
LIN {X 0,Y 594.383,Z 331.448,A -85,B 0,C 180,E1 -1033.84,E2 -1033.84} C_VEL
LIN {X 0,Y 594.367,Z 331.451,A -85,B 0,C 180,E1 -1036.7,E2 -1036.7} C_VEL
LIN {X 0,Y 594.374,Z 331.452,A -85,B 0,C 180,E1 -1039.433,E2 -1039.433} C_VEL
LIN {X 0,Y 594.391,Z 331.449,A -85,B 0,C 180,E1 -1042.391,E2 -1042.391} C_VEL
LIN {X 0,Y 594.388,Z 331.448,A -85,B 0,C 180,E1 -1044.671,E2 -1044.671} C_VEL
LIN {X 0,Y 594.379,Z 331.449,A -85,B 0,C 180,E1 -1047.088,E2 -1047.088} C_VEL
LIN {X 0,Y 594.401,Z 331.444,A -85,B 0,C 180,E1 -1049.669,E2 -1049.669} C_VEL
LIN {X 0,Y 594.39,Z 331.448,A -85,B 0,C 180,E1 -1052.54,E2 -1052.54} C_VEL
LIN {X 0,Y 594.382,Z 331.448,A -85,B 0,C 180,E1 -1054.807,E2 -1054.807} C_VEL
LIN {X 0,Y 594.366,Z 331.451,A -85,B 0,C 180,E1 -1057.263,E2 -1057.263} C_VEL
LIN {X 0,Y 594.381,Z 331.448,A -85,B 0,C 180,E1 -1059.946,E2 -1059.946} C_VEL
LIN {X 0,Y 594.394,Z 331.446,A -85,B 0,C 180,E1 -1062.806,E2 -1062.806} C_VEL
LIN {X 0,Y 594.387,Z 331.448,A -85,B 0,C 180,E1 -1065.825,E2 -1065.825} C_VEL
LIN {X 0,Y 594.394,Z 331.449,A -85,B 0,C 180,E1 -1068.404,E2 -1068.404} C_VEL
LIN {X 0,Y 594.403,Z 331.447,A -85,B 0,C 180,E1 -1071.158,E2 -1071.158} C_VEL
LIN {X 0,Y 594.366,Z 331.45,A -85,B 0,C 180,E1 -1073.891,E2 -1073.891} C_VEL
LIN {X 0,Y 594.384,Z 331.448,A -85,B 0,C 180,E1 -1076.611,E2 -1076.611} C_VEL
LIN {X 0,Y 594.428,Z 331.444,A -85,B 0,C 180,E1 -1079.322,E2 -1079.322} C_VEL
LIN {X 0,Y 594.392,Z 331.448,A -85,B 0,C 180,E1 -1082.033,E2 -1082.033} C_VEL
LIN {X 0,Y 594.394,Z 331.446,A -85,B 0,C 180,E1 -1084.747,E2 -1084.747} C_VEL
LIN {X 0,Y 594.4,Z 331.447,A -85,B 0,C 180,E1 -1087.473,E2 -1087.473} C_VEL
LIN {X 0,Y 594.39,Z 331.449,A -85,B 0,C 180,E1 -1090.216,E2 -1090.216} C_VEL
LIN {X 0,Y 594.37,Z 331.45,A -85,B 0,C 180,E1 -1092.983,E2 -1092.983} C_VEL
LIN {X 0,Y 594.365,Z 331.45,A -85,B 0,C 180,E1 -1095.781,E2 -1095.781} C_VEL
LIN {X 0,Y 594.381,Z 331.448,A -85,B 0,C 180,E1 -1098.618,E2 -1098.618} C_VEL
LIN {X 0,Y 594.366,Z 331.451,A -85,B 0,C 180,E1 -1101.503,E2 -1101.503} C_VEL
LIN {X 0,Y 594.386,Z 331.449,A -85,B 0,C 180,E1 -1104.446,E2 -1104.446} C_VEL
LIN {X 0,Y 594.388,Z 331.448,A -85,B 0,C 180,E1 -1106.699,E2 -1106.699} C_VEL
LIN {X 0,Y 594.379,Z 331.45,A -85,B 0,C 180,E1 -1108.999,E2 -1108.999} C_VEL
LIN {X 0,Y 594.392,Z 331.447,A -85,B 0,C 180,E1 -1111.646,E2 -1111.646} C_VEL
LIN {X 0,Y 594.395,Z 331.447,A -85,B 0,C 180,E1 -1114.579,E2 -1114.579} C_VEL
LIN {X 0,Y 594.387,Z 331.45,A -85,B 0,C 180,E1 -1117.087,E2 -1117.087} C_VEL
LIN {X 0,Y 594.38,Z 331.449,A -85,B 0,C 180,E1 -1119.776,E2 -1119.776} C_VEL
LIN {X 0,Y 594.37,Z 331.451,A -85,B 0,C 180,E1 -1122.375,E2 -1122.375} C_VEL
LIN {X 0,Y 594.362,Z 331.453,A -85,B 0,C 180,E1 -1125.192,E2 -1125.192} C_VEL
LIN {X 0,Y 594.389,Z 331.448,A -85,B 0,C 180,E1 -1127.627,E2 -1127.627} C_VEL
LIN {X 0,Y 594.396,Z 331.448,A -85,B 0,C 180,E1 -1130.322,E2 -1130.322} C_VEL
LIN {X 0,Y 594.389,Z 331.449,A -85,B 0,C 180,E1 -1132.914,E2 -1132.914} C_VEL
LIN {X 0,Y 594.424,Z 331.59,A -85,B 0,C 180,E1 -1134.076,E2 -1134.076} C_VEL
LIN {X 0,Y 594.766,Z 335.939,A -85,B 0,C 180,E1 -1135.036,E2 -1135.036} C_VEL
LIN {X 0,Y 594.644,Z 350.688,A -85,B 0,C 180,E1 -1138.133,E2 -1138.133} C_VEL
LIN {X 0,Y 594.725,Z 363.128,A -85,B 0,C 180,E1 -1140.633,E2 -1140.633} C_VEL
LIN {X 0,Y 594.683,Z 375.961,A -85,B 0,C 180,E1 -1143.316,E2 -1143.316} C_VEL
LIN {X 0,Y 594.585,Z 390.488,A -85,B 0,C 180,E1 -1146.305,E2 -1146.305} C_VEL
LIN {X 0,Y 594.512,Z 404.124,A -85,B 0,C 180,E1 -1149.051,E2 -1149.051} C_VEL
LIN {X 0,Y 594.438,Z 417.726,A -85,B 0,C 180,E1 -1151.742,E2 -1151.742} C_VEL
LIN {X 0,Y 594.391,Z 432.253,A -85,B 0,C 180,E1 -1154.572,E2 -1154.572} C_VEL
LIN {X 0,Y 594.346,Z 446.78,A -85,B 0,C 180,E1 -1157.364,E2 -1157.364} C_VEL
LIN {X 0,Y 594.39,Z 449.882,A -85,B 0,C 180,E1 -1157.918,E2 -1157.918} C_VEL
LIN {X 0,Y 594.676,Z 457.257,A -85,B 0,C 180,E1 -1158.043,E2 -1158.043} C_VEL
LIN {X 0,Y 594.625,Z 470.514,A -85,B 0,C 180,E1 -1158.366,E2 -1158.366} C_VEL
LIN {X 0,Y 594.562,Z 482.718,A -85,B 0,C 180,E1 -1158.805,E2 -1158.805} C_VEL
LIN {X 0,Y 594.515,Z 494.218,A -85,B 0,C 180,E1 -1159.356,E2 -1159.356} C_VEL
LIN {X 0,Y 594.475,Z 505.484,A -85,B 0,C 180,E1 -1160.044,E2 -1160.044} C_VEL
LIN {X 0,Y 594.406,Z 515.653,A -85,B 0,C 180,E1 -1160.816,E2 -1160.816} C_VEL
LIN {X 0,Y 594.372,Z 524.792,A -85,B 0,C 180,E1 -1161.672,E2 -1161.672} C_VEL
LIN {X 0,Y 594.316,Z 533.695,A -85,B 0,C 180,E1 -1162.697,E2 -1162.697} C_VEL
LIN {X 0,Y 594.281,Z 540.169,A -85,B 0,C 180,E1 -1163.615,E2 -1163.615} C_VEL
LIN {X 0,Y 594.289,Z 545.683,A -85,B 0,C 180,E1 -1164.572,E2 -1164.572} C_VEL
LIN {X 0,Y 594.27,Z 550.373,A -85,B 0,C 180,E1 -1165.592,E2 -1165.592} C_VEL
LIN {X 0,Y 594.267,Z 553.958,A -85,B 0,C 180,E1 -1166.611,E2 -1166.611} C_VEL
LIN {X 0,Y 594.226,Z 555.81,A -85,B 0,C 180,E1 -1167.289,E2 -1167.289} C_VEL
LIN {X 0,Y 594.242,Z 557.202,A -85,B 0,C 180,E1 -1167.967,E2 -1167.967} C_VEL
LIN {X 0,Y 594.239,Z 558.784,A -85,B 0,C 180,E1 -1169.323,E2 -1169.323} C_VEL
LIN {X 0,Y 594.236,Z 559,A -85,B 0,C 180,E1 -1170,E2 -1170} C_VEL
LIN {X 0,Y 594.248,Z 558.184,A -85,B 0,C 180,E1 -1171.356,E2 -1171.356} C_VEL
LIN {X 0,Y 594.242,Z 557.201,A -85,B 0,C 180,E1 -1172.034,E2 -1172.034} C_VEL
LIN {X 0,Y 594.226,Z 555.808,A -85,B 0,C 180,E1 -1172.712,E2 -1172.712} C_VEL
LIN {X 0,Y 594.288,Z 552.894,A -85,B 0,C 180,E1 -1173.73,E2 -1173.73} C_VEL
LIN {X 0,Y 594.241,Z 548.948,A -85,B 0,C 180,E1 -1174.749,E2 -1174.749} C_VEL
LIN {X 0,Y 594.304,Z 542.874,A -85,B 0,C 180,E1 -1175.94,E2 -1175.94} C_VEL
LIN {X 0,Y 594.308,Z 536.232,A -85,B 0,C 180,E1 -1176.963,E2 -1176.963} C_VEL
LIN {X 0,Y 594.359,Z 527.985,A -85,B 0,C 180,E1 -1177.987,E2 -1177.987} C_VEL
LIN {X 0,Y 594.382,Z 519.532,A -85,B 0,C 180,E1 -1178.843,E2 -1178.843} C_VEL
LIN {X 0,Y 594.435,Z 509.087,A -85,B 0,C 180,E1 -1179.7,E2 -1179.7} C_VEL
LIN {X 0,Y 594.482,Z 498.75,A -85,B 0,C 180,E1 -1180.387,E2 -1180.387} C_VEL
LIN {X 0,Y 594.557,Z 487.735,A -85,B 0,C 180,E1 -1180.973,E2 -1180.973} C_VEL
LIN {X 0,Y 594.583,Z 475.702,A -85,B 0,C 180,E1 -1181.464,E2 -1181.464} C_VEL
LIN {X 0,Y 594.644,Z 462.33,A -85,B 0,C 180,E1 -1181.851,E2 -1181.851} C_VEL
LIN {X 0,Y 594.465,Z 450.566,A -85,B 0,C 180,E1 -1182.071,E2 -1182.071} C_VEL
LIN {X 0,Y 594.364,Z 449.498,A -85,B 0,C 180,E1 -1182.116,E2 -1182.116} C_VEL
LIN {X 0,Y 594.386,Z 435.879,A -85,B 0,C 180,E1 -1184.728,E2 -1184.728} C_VEL
LIN {X 0,Y 594.424,Z 421.353,A -85,B 0,C 180,E1 -1187.548,E2 -1187.548} C_VEL
LIN {X 0,Y 594.472,Z 408.642,A -85,B 0,C 180,E1 -1190.051,E2 -1190.051} C_VEL
LIN {X 0,Y 594.561,Z 395.004,A -85,B 0,C 180,E1 -1192.78,E2 -1192.78} C_VEL
LIN {X 0,Y 594.631,Z 381.404,A -85,B 0,C 180,E1 -1195.557,E2 -1195.557} C_VEL
LIN {X 0,Y 594.72,Z 368.693,A -85,B 0,C 180,E1 -1198.21,E2 -1198.21} C_VEL
LIN {X 0,Y 594.71,Z 357.318,A -85,B 0,C 180,E1 -1200.541,E2 -1200.541} C_VEL
LIN {X 0,Y 594.684,Z 343.661,A -85,B 0,C 180,E1 -1203.336,E2 -1203.336} C_VEL
LIN {X 0,Y 594.748,Z 334.13,A -85,B 0,C 180,E1 -1205.382,E2 -1205.382} C_VEL
LIN {X 0,Y 594.377,Z 331.452,A -85,B 0,C 180,E1 -1206.034,E2 -1206.034} C_VEL
LIN {X 0,Y 594.374,Z 331.449,A -85,B 0,C 180,E1 -1208.806,E2 -1208.806} C_VEL
LIN {X 0,Y 594.388,Z 331.449,A -85,B 0,C 180,E1 -1211.849,E2 -1211.849} C_VEL
LIN {X 0,Y 594.387,Z 331.448,A -85,B 0,C 180,E1 -1214.236,E2 -1214.236} C_VEL
LIN {X 0,Y 594.362,Z 331.452,A -85,B 0,C 180,E1 -1217.149,E2 -1217.149} C_VEL
LIN {X 0,Y 594.375,Z 331.451,A -85,B 0,C 180,E1 -1219.433,E2 -1219.433} C_VEL
LIN {X 0,Y 594.397,Z 331.446,A -85,B 0,C 180,E1 -1222.392,E2 -1222.392} C_VEL
LIN {X 0,Y 594.387,Z 331.448,A -85,B 0,C 180,E1 -1225.42,E2 -1225.42} C_VEL
LIN {X 0,Y 594.398,Z 331.447,A -85,B 0,C 180,E1 -1228.355,E2 -1228.355} C_VEL
LIN {X 0,Y 594.387,Z 331.448,A -85,B 0,C 180,E1 -1231.043,E2 -1231.043} C_VEL
LIN {X 0,Y 594.387,Z 331.447,A -85,B 0,C 180,E1 -1233.301,E2 -1233.301} C_VEL
LIN {X 0,Y 594.398,Z 331.448,A -85,B 0,C 180,E1 -1236.296,E2 -1236.296} C_VEL
LIN {X 0,Y 594.402,Z 331.445,A -85,B 0,C 180,E1 -1239.224,E2 -1239.224} C_VEL
LIN {X 0,Y 594.352,Z 331.453,A -85,B 0,C 180,E1 -1242.095,E2 -1242.095} C_VEL
LIN {X 0,Y 594.375,Z 331.452,A -85,B 0,C 180,E1 -1244.219,E2 -1244.219} C_VEL
LIN {X 0,Y 594.389,Z 331.449,A -85,B 0,C 180,E1 -1246.321,E2 -1246.321} C_VEL
LIN {X 0,Y 594.376,Z 331.448,A -85,B 0,C 180,E1 -1249.095,E2 -1249.095} C_VEL
LIN {X 0,Y 594.42,Z 331.444,A -85,B 0,C 180,E1 -1251.843,E2 -1251.843} C_VEL
LIN {X 0,Y 594.396,Z 331.447,A -85,B 0,C 180,E1 -1254.572,E2 -1254.572} C_VEL
LIN {X 0,Y 594.411,Z 331.444,A -85,B 0,C 180,E1 -1257.289,E2 -1257.289} C_VEL
LIN {X 0,Y 594.42,Z 331.445,A -85,B 0,C 180,E1 -1260,E2 -1260} C_VEL
LIN {X 0,Y 594.412,Z 331.444,A -85,B 0,C 180,E1 -1262.711,E2 -1262.711} C_VEL
LIN {X 0,Y 594.394,Z 331.449,A -85,B 0,C 180,E1 -1265.428,E2 -1265.428} C_VEL
LIN {X 0,Y 594.421,Z 331.443,A -85,B 0,C 180,E1 -1268.157,E2 -1268.157} C_VEL
LIN {X 0,Y 594.393,Z 331.449,A -85,B 0,C 180,E1 -1271.073,E2 -1271.073} C_VEL
LIN {X 0,Y 594.385,Z 331.448,A -85,B 0,C 180,E1 -1273.679,E2 -1273.679} C_VEL
LIN {X 0,Y 594.367,Z 331.449,A -85,B 0,C 180,E1 -1275.328,E2 -1275.328} C_VEL
LIN {X 0,Y 593.696,Z 331.534,A -85,B 0,C 180,E1 -1275.894,E2 -1275.894} C_VEL
LIN {X 0,Y 590.843,Z 331.891,A -85,B 0,C 180,E1 -1276.812,E2 -1276.812} C_VEL
LIN {X 0,Y 588.437,Z 332.19,A -85,B 0,C 180,E1 -1277.551,E2 -1277.551} C_VEL
LIN {X 0,Y 587.409,Z 332.317,A -85,B 0,C 180,E1 -1278.121,E2 -1278.121} C_VEL
LIN {X 0,Y 587.328,Z 332.326,A -85,B 0,C 180,E1 -1278.314,E2 -1278.314} C_VEL
LIN {X 0,Y 587.338,Z 332.326,A -85,B 0,C 180,E1 -1281.038,E2 -1281.038} C_VEL
LIN {X 0,Y 587.329,Z 332.327,A -85,B 0,C 180,E1 -1283.259,E2 -1283.259} C_VEL
LIN {X 0,Y 587.343,Z 332.326,A -85,B 0,C 180,E1 -1285.517,E2 -1285.517} C_VEL
LIN {X 0,Y 587.352,Z 332.326,A -85,B 0,C 180,E1 -1287.818,E2 -1287.818} C_VEL
LIN {X 0,Y 587.344,Z 332.324,A -85,B 0,C 180,E1 -1290.51,E2 -1290.51} C_VEL
LIN {X 0,Y 587.343,Z 332.326,A -85,B 0,C 180,E1 -1293.397,E2 -1293.397} C_VEL
LIN {X 0,Y 587.298,Z 332.332,A -85,B 0,C 180,E1 -1295.9,E2 -1295.9} C_VEL
LIN {X 0,Y 587.34,Z 332.325,A -85,B 0,C 180,E1 -1298.479,E2 -1298.479} C_VEL
LIN {X 0,Y 587.343,Z 332.325,A -85,B 0,C 180,E1 -1301.157,E2 -1301.157} C_VEL
LIN {X 0,Y 587.318,Z 332.327,A -85,B 0,C 180,E1 -1304.112,E2 -1304.112} C_VEL
LIN {X 0,Y 587.33,Z 332.329,A -85,B 0,C 180,E1 -1306.994,E2 -1306.994} C_VEL
LIN {X 0,Y 587.319,Z 332.327,A -85,B 0,C 180,E1 -1309.745,E2 -1309.745} C_VEL
LIN {X 0,Y 587.348,Z 332.325,A -85,B 0,C 180,E1 -1312.392,E2 -1312.392} C_VEL
LIN {X 0,Y 587.367,Z 332.323,A -85,B 0,C 180,E1 -1315.78,E2 -1315.78} C_VEL
LIN {X 0,Y 587.349,Z 332.326,A -85,B 0,C 180,E1 -1318.231,E2 -1318.231} C_VEL
LIN {X 0,Y 587.355,Z 332.323,A -85,B 0,C 180,E1 -1320.867,E2 -1320.867} C_VEL
LIN {X 0,Y 587.367,Z 332.324,A -85,B 0,C 180,E1 -1323.819,E2 -1323.819} C_VEL
LIN {X 0,Y 587.342,Z 332.327,A -85,B 0,C 180,E1 -1325.993,E2 -1325.993} C_VEL
LIN {X 0,Y 587.324,Z 332.329,A -85,B 0,C 180,E1 -1328.225,E2 -1328.225} C_VEL
LIN {X 0,Y 587.357,Z 332.323,A -85,B 0,C 180,E1 -1331.151,E2 -1331.151} C_VEL
LIN {X 0,Y 587.33,Z 332.328,A -85,B 0,C 180,E1 -1334.024,E2 -1334.024} C_VEL
LIN {X 0,Y 587.365,Z 332.325,A -85,B 0,C 180,E1 -1336.154,E2 -1336.154} C_VEL
LIN {X 0,Y 587.35,Z 332.324,A -85,B 0,C 180,E1 -1338.962,E2 -1338.962} C_VEL
LIN {X 0,Y 587.372,Z 332.324,A -85,B 0,C 180,E1 -1341.744,E2 -1341.744} C_VEL
LIN {X 0,Y 587.358,Z 332.323,A -85,B 0,C 180,E1 -1344.507,E2 -1344.507} C_VEL
LIN {X 0,Y 587.347,Z 332.326,A -85,B 0,C 180,E1 -1346.033,E2 -1346.033} C_VEL
LIN {X 0,Y 587.667,Z 336.022,A -85,B 0,C 180,E1 -1346.142,E2 -1346.142} C_VEL
LIN {X 0,Y 587.612,Z 349.115,A -85,B 0,C 180,E1 -1346.571,E2 -1346.571} C_VEL
LIN {X 0,Y 587.539,Z 360.668,A -85,B 0,C 180,E1 -1347.085,E2 -1347.085} C_VEL
LIN {X 0,Y 587.504,Z 371.221,A -85,B 0,C 180,E1 -1347.686,E2 -1347.686} C_VEL
LIN {X 0,Y 587.418,Z 382.074,A -85,B 0,C 180,E1 -1348.457,E2 -1348.457} C_VEL
LIN {X 0,Y 587.324,Z 391.794,A -85,B 0,C 180,E1 -1349.314,E2 -1349.314} C_VEL
LIN {X 0,Y 587.271,Z 401.244,A -85,B 0,C 180,E1 -1350.342,E2 -1350.342} C_VEL
LIN {X 0,Y 587.208,Z 408.798,A -85,B 0,C 180,E1 -1351.371,E2 -1351.371} C_VEL
LIN {X 0,Y 587.193,Z 414.891,A -85,B 0,C 180,E1 -1352.4,E2 -1352.4} C_VEL
LIN {X 0,Y 587.198,Z 419.74,A -85,B 0,C 180,E1 -1353.43,E2 -1353.43} C_VEL
LIN {X 0,Y 587.186,Z 423.488,A -85,B 0,C 180,E1 -1354.462,E2 -1354.462} C_VEL
LIN {X 0,Y 587.179,Z 426.228,A -85,B 0,C 180,E1 -1355.494,E2 -1355.494} C_VEL
LIN {X 0,Y 587.168,Z 428.413,A -85,B 0,C 180,E1 -1356.874,E2 -1356.874} C_VEL
LIN {X 0,Y 587.146,Z 428.897,A -85,B 0,C 180,E1 -1357.565,E2 -1357.565} C_VEL
LIN {X 0,Y 587.127,Z 428.634,A -85,B 0,C 180,E1 -1358.952,E2 -1358.952} C_VEL
LIN {X 0,Y 587.151,Z 427.919,A -85,B 0,C 180,E1 -1359.646,E2 -1359.646} C_VEL
LIN {X 0,Y 587.14,Z 426.755,A -85,B 0,C 180,E1 -1360.343,E2 -1360.343} C_VEL
LIN {X 0,Y 587.15,Z 424.221,A -85,B 0,C 180,E1 -1361.39,E2 -1361.39} C_VEL
LIN {X 0,Y 587.181,Z 420.644,A -85,B 0,C 180,E1 -1362.441,E2 -1362.441} C_VEL
LIN {X 0,Y 587.197,Z 415.907,A -85,B 0,C 180,E1 -1363.496,E2 -1363.496} C_VEL
LIN {X 0,Y 587.22,Z 409.854,A -85,B 0,C 180,E1 -1364.556,E2 -1364.556} C_VEL
LIN {X 0,Y 587.26,Z 402.249,A -85,B 0,C 180,E1 -1365.62,E2 -1365.62} C_VEL
LIN {X 0,Y 587.318,Z 394.447,A -85,B 0,C 180,E1 -1366.51,E2 -1366.51} C_VEL
LIN {X 0,Y 587.407,Z 384.882,A -85,B 0,C 180,E1 -1367.404,E2 -1367.404} C_VEL
LIN {X 0,Y 587.448,Z 374.149,A -85,B 0,C 180,E1 -1368.212,E2 -1368.212} C_VEL
LIN {X 0,Y 587.571,Z 362.367,A -85,B 0,C 180,E1 -1368.918,E2 -1368.918} C_VEL
LIN {X 0,Y 587.588,Z 349.942,A -85,B 0,C 180,E1 -1369.487,E2 -1369.487} C_VEL
LIN {X 0,Y 587.704,Z 336.757,A -85,B 0,C 180,E1 -1369.926,E2 -1369.926} C_VEL
LIN {X 0,Y 587.444,Z 332.857,A -85,B 0,C 180,E1 -1370.03,E2 -1370.03} C_VEL
LIN {X 0,Y 587.356,Z 332.324,A -85,B 0,C 180,E1 -1370.075,E2 -1370.075} C_VEL
LIN {X 0,Y 587.321,Z 332.328,A -85,B 0,C 180,E1 -1372.868,E2 -1372.868} C_VEL
LIN {X 0,Y 587.337,Z 332.328,A -85,B 0,C 180,E1 -1375.516,E2 -1375.516} C_VEL
LIN {X 0,Y 587.343,Z 332.326,A -85,B 0,C 180,E1 -1377.817,E2 -1377.817} C_VEL
LIN {X 0,Y 587.337,Z 332.329,A -85,B 0,C 180,E1 -1380.509,E2 -1380.509} C_VEL
LIN {X 0,Y 587.339,Z 332.327,A -85,B 0,C 180,E1 -1383.396,E2 -1383.396} C_VEL
LIN {X 0,Y 587.294,Z 332.332,A -85,B 0,C 180,E1 -1385.899,E2 -1385.899} C_VEL
LIN {X 0,Y 587.33,Z 332.329,A -85,B 0,C 180,E1 -1388.479,E2 -1388.479} C_VEL
LIN {X 0,Y 587.339,Z 332.326,A -85,B 0,C 180,E1 -1391.156,E2 -1391.156} C_VEL
LIN {X 0,Y 587.335,Z 332.326,A -85,B 0,C 180,E1 -1394.114,E2 -1394.114} C_VEL
LIN {X 0,Y 587.315,Z 332.328,A -85,B 0,C 180,E1 -1396.993,E2 -1396.993} C_VEL
LIN {X 0,Y 587.321,Z 332.328,A -85,B 0,C 180,E1 -1399.746,E2 -1399.746} C_VEL
LIN {X 0,Y 587.346,Z 332.327,A -85,B 0,C 180,E1 -1402.392,E2 -1402.392} C_VEL
LIN {X 0,Y 587.353,Z 332.324,A -85,B 0,C 180,E1 -1404.946,E2 -1404.946} C_VEL
LIN {X 0,Y 587.34,Z 332.327,A -85,B 0,C 180,E1 -1407.421,E2 -1407.421} C_VEL
LIN {X 0,Y 587.347,Z 332.321,A -85,B 0,C 180,E1 -1409.83,E2 -1409.83} C_VEL
LIN {X 0,Y 587.351,Z 332.325,A -85,B 0,C 180,E1 -1412.306,E2 -1412.306} C_VEL
LIN {X 0,Y 587.341,Z 332.327,A -85,B 0,C 180,E1 -1414.483,E2 -1414.483} C_VEL
LIN {X 0,Y 587.32,Z 332.327,A -85,B 0,C 180,E1 -1417.13,E2 -1417.13} C_VEL
LIN {X 0,Y 587.335,Z 332.326,A -85,B 0,C 180,E1 -1419.695,E2 -1419.695} C_VEL
LIN {X 0,Y 587.36,Z 332.323,A -85,B 0,C 180,E1 -1422.594,E2 -1422.594} C_VEL
LIN {X 0,Y 587.363,Z 332.323,A -85,B 0,C 180,E1 -1425.739,E2 -1425.739} C_VEL
LIN {X 0,Y 587.361,Z 332.323,A -85,B 0,C 180,E1 -1428.858,E2 -1428.858} C_VEL
LIN {X 0,Y 587.371,Z 332.322,A -85,B 0,C 180,E1 -1431.745,E2 -1431.745} C_VEL
LIN {X 0,Y 587.359,Z 332.323,A -85,B 0,C 180,E1 -1434.507,E2 -1434.507} C_VEL
LIN {X 0,Y 587.38,Z 332.323,A -85,B 0,C 180,E1 -1437.257,E2 -1437.257} C_VEL
LIN {X 0,Y 587.381,Z 332.32,A -85,B 0,C 180,E1 -1440,E2 -1440} C_VEL
LIN {X 0,Y 587.377,Z 332.321,A -85,B 0,C 180,E1 -1442.743,E2 -1442.743} C_VEL
LIN {X 0,Y 587.362,Z 332.323,A -85,B 0,C 180,E1 -1445.493,E2 -1445.493} C_VEL
LIN {X 0,Y 587.367,Z 332.325,A -85,B 0,C 180,E1 -1448.255,E2 -1448.255} C_VEL
LIN {X 0,Y 587.344,Z 332.326,A -85,B 0,C 180,E1 -1451.134,E2 -1451.134} C_VEL
LIN {X 0,Y 587.362,Z 332.325,A -85,B 0,C 180,E1 -1454.261,E2 -1454.261} C_VEL
LIN {X 0,Y 587.355,Z 332.324,A -85,B 0,C 180,E1 -1457.406,E2 -1457.406} C_VEL
LIN {X 0,Y 587.327,Z 332.328,A -85,B 0,C 180,E1 -1460.305,E2 -1460.305} C_VEL
LIN {X 0,Y 587.321,Z 332.33,A -85,B 0,C 180,E1 -1463.259,E2 -1463.259} C_VEL
LIN {X 0,Y 587.334,Z 332.327,A -85,B 0,C 180,E1 -1465.517,E2 -1465.517} C_VEL
LIN {X 0,Y 587.346,Z 332.325,A -85,B 0,C 180,E1 -1467.818,E2 -1467.818} C_VEL
LIN {X 0,Y 587.35,Z 332.325,A -85,B 0,C 180,E1 -1470.513,E2 -1470.513} C_VEL
LIN {X 0,Y 587.335,Z 332.327,A -85,B 0,C 180,E1 -1473.397,E2 -1473.397} C_VEL
LIN {X 0,Y 587.355,Z 332.324,A -85,B 0,C 180,E1 -1475.896,E2 -1475.896} C_VEL
LIN {X 0,Y 587.336,Z 332.325,A -85,B 0,C 180,E1 -1478.479,E2 -1478.479} C_VEL
LIN {X 0,Y 587.362,Z 332.324,A -85,B 0,C 180,E1 -1481.155,E2 -1481.155} C_VEL
LIN {X 0,Y 587.333,Z 332.328,A -85,B 0,C 180,E1 -1484.115,E2 -1484.115} C_VEL
LIN {X 0,Y 587.336,Z 332.327,A -85,B 0,C 180,E1 -1486.996,E2 -1486.996} C_VEL
LIN {X 0,Y 587.33,Z 332.327,A -85,B 0,C 180,E1 -1489.748,E2 -1489.748} C_VEL
LIN {X 0,Y 587.348,Z 332.326,A -85,B 0,C 180,E1 -1492.393,E2 -1492.393} C_VEL
LIN {X 0,Y 587.368,Z 332.41,A -85,B 0,C 180,E1 -1493.868,E2 -1493.868} C_VEL
LIN {X 0,Y 587.844,Z 337.367,A -85,B 0,C 180,E1 -1494.98,E2 -1494.98} C_VEL
LIN {X 0,Y 587.68,Z 352.076,A -85,B 0,C 180,E1 -1498.112,E2 -1498.112} C_VEL
LIN {X 0,Y 587.74,Z 365.299,A -85,B 0,C 180,E1 -1500.799,E2 -1500.799} C_VEL
LIN {X 0,Y 587.769,Z 375.961,A -85,B 0,C 180,E1 -1502.976,E2 -1502.976} C_VEL
LIN {X 0,Y 587.63,Z 388.926,A -85,B 0,C 180,E1 -1505.684,E2 -1505.684} C_VEL
LIN {X 0,Y 587.55,Z 403.201,A -85,B 0,C 180,E1 -1508.604,E2 -1508.604} C_VEL
LIN {X 0,Y 587.442,Z 417.726,A -85,B 0,C 180,E1 -1511.517,E2 -1511.517} C_VEL
LIN {X 0,Y 587.346,Z 430.437,A -85,B 0,C 180,E1 -1514.026,E2 -1514.026} C_VEL
LIN {X 0,Y 587.338,Z 443.148,A -85,B 0,C 180,E1 -1516.507,E2 -1516.507} C_VEL
LIN {X 0,Y 587.336,Z 449.882,A -85,B 0,C 180,E1 -1517.771,E2 -1517.771} C_VEL
LIN {X 0,Y 587.745,Z 454.973,A -85,B 0,C 180,E1 -1517.856,E2 -1517.856} C_VEL
LIN {X 0,Y 587.672,Z 468.236,A -85,B 0,C 180,E1 -1518.161,E2 -1518.161} C_VEL
LIN {X 0,Y 587.623,Z 480.645,A -85,B 0,C 180,E1 -1518.586,E2 -1518.586} C_VEL
LIN {X 0,Y 587.559,Z 492.641,A -85,B 0,C 180,E1 -1519.142,E2 -1519.142} C_VEL
LIN {X 0,Y 587.466,Z 504.208,A -85,B 0,C 180,E1 -1519.837,E2 -1519.837} C_VEL
LIN {X 0,Y 587.366,Z 514.603,A -85,B 0,C 180,E1 -1520.618,E2 -1520.618} C_VEL
LIN {X 0,Y 587.321,Z 523.117,A -85,B 0,C 180,E1 -1521.398,E2 -1521.398} C_VEL
LIN {X 0,Y 587.273,Z 530.965,A -85,B 0,C 180,E1 -1522.263,E2 -1522.263} C_VEL
LIN {X 0,Y 587.23,Z 537.473,A -85,B 0,C 180,E1 -1523.127,E2 -1523.127} C_VEL
LIN {X 0,Y 587.236,Z 543.869,A -85,B 0,C 180,E1 -1524.162,E2 -1524.162} C_VEL
LIN {X 0,Y 587.147,Z 548.952,A -85,B 0,C 180,E1 -1525.194,E2 -1525.194} C_VEL
LIN {X 0,Y 587.212,Z 552.897,A -85,B 0,C 180,E1 -1526.226,E2 -1526.226} C_VEL
LIN {X 0,Y 587.132,Z 555.81,A -85,B 0,C 180,E1 -1527.256,E2 -1527.256} C_VEL
LIN {X 0,Y 587.141,Z 557.201,A -85,B 0,C 180,E1 -1527.943,E2 -1527.943} C_VEL
LIN {X 0,Y 587.14,Z 558.785,A -85,B 0,C 180,E1 -1529.315,E2 -1529.315} C_VEL
LIN {X 0,Y 587.137,Z 559,A -85,B 0,C 180,E1 -1530,E2 -1530} C_VEL
LIN {X 0,Y 587.147,Z 558.185,A -85,B 0,C 180,E1 -1531.372,E2 -1531.372} C_VEL
LIN {X 0,Y 587.141,Z 557.2,A -85,B 0,C 180,E1 -1532.058,E2 -1532.058} C_VEL
LIN {X 0,Y 587.132,Z 555.808,A -85,B 0,C 180,E1 -1532.745,E2 -1532.745} C_VEL
LIN {X 0,Y 587.212,Z 552.894,A -85,B 0,C 180,E1 -1533.775,E2 -1533.775} C_VEL
LIN {X 0,Y 587.147,Z 548.947,A -85,B 0,C 180,E1 -1534.807,E2 -1534.807} C_VEL
LIN {X 0,Y 587.217,Z 542.875,A -85,B 0,C 180,E1 -1536.012,E2 -1536.012} C_VEL
LIN {X 0,Y 587.245,Z 536.233,A -85,B 0,C 180,E1 -1537.047,E2 -1537.047} C_VEL
LIN {X 0,Y 587.3,Z 527.986,A -85,B 0,C 180,E1 -1538.084,E2 -1538.084} C_VEL
LIN {X 0,Y 587.344,Z 519.532,A -85,B 0,C 180,E1 -1538.949,E2 -1538.949} C_VEL
LIN {X 0,Y 587.422,Z 509.088,A -85,B 0,C 180,E1 -1539.817,E2 -1539.817} C_VEL
LIN {X 0,Y 587.486,Z 498.75,A -85,B 0,C 180,E1 -1540.512,E2 -1540.512} C_VEL
LIN {X 0,Y 587.561,Z 486.81,A -85,B 0,C 180,E1 -1541.149,E2 -1541.149} C_VEL
LIN {X 0,Y 587.633,Z 474.586,A -85,B 0,C 180,E1 -1541.64,E2 -1541.64} C_VEL
LIN {X 0,Y 587.713,Z 461.415,A -85,B 0,C 180,E1 -1542.014,E2 -1542.014} C_VEL
LIN {X 0,Y 587.622,Z 451.884,A -85,B 0,C 180,E1 -1542.194,E2 -1542.194} C_VEL
LIN {X 0,Y 587.318,Z 449.612,A -85,B 0,C 180,E1 -1542.242,E2 -1542.242} C_VEL
LIN {X 0,Y 587.352,Z 435.879,A -85,B 0,C 180,E1 -1544.908,E2 -1544.908} C_VEL
LIN {X 0,Y 587.411,Z 421.353,A -85,B 0,C 180,E1 -1547.764,E2 -1547.764} C_VEL
LIN {X 0,Y 587.516,Z 406.826,A -85,B 0,C 180,E1 -1550.664,E2 -1550.664} C_VEL
LIN {X 0,Y 587.621,Z 392.299,A -85,B 0,C 180,E1 -1553.62,E2 -1553.62} C_VEL
LIN {X 0,Y 587.753,Z 377.772,A -85,B 0,C 180,E1 -1556.642,E2 -1556.642} C_VEL
LIN {X 0,Y 587.746,Z 366.883,A -85,B 0,C 180,E1 -1558.888,E2 -1558.888} C_VEL
LIN {X 0,Y 587.719,Z 354.807,A -85,B 0,C 180,E1 -1561.345,E2 -1561.345} C_VEL
LIN {X 0,Y 587.767,Z 343.216,A -85,B 0,C 180,E1 -1563.781,E2 -1563.781} C_VEL
LIN {X 0,Y 587.76,Z 334.89,A -85,B 0,C 180,E1 -1565.6,E2 -1565.6} C_VEL
LIN {X 0,Y 587.329,Z 332.329,A -85,B 0,C 180,E1 -1566.216,E2 -1566.216} C_VEL
LIN {X 0,Y 587.32,Z 332.328,A -85,B 0,C 180,E1 -1568.94,E2 -1568.94} C_VEL
LIN {X 0,Y 587.358,Z 332.323,A -85,B 0,C 180,E1 -1572.073,E2 -1572.073} C_VEL
LIN {X 0,Y 587.322,Z 332.33,A -85,B 0,C 180,E1 -1575.089,E2 -1575.089} C_VEL
LIN {X 0,Y 587.326,Z 332.326,A -85,B 0,C 180,E1 -1577.925,E2 -1577.925} C_VEL
LIN {X 0,Y 587.352,Z 332.326,A -85,B 0,C 180,E1 -1580.641,E2 -1580.641} C_VEL
LIN {X 0,Y 587.353,Z 332.323,A -85,B 0,C 180,E1 -1583.293,E2 -1583.293} C_VEL
LIN {X 0,Y 587.367,Z 332.321,A -85,B 0,C 180,E1 -1585.78,E2 -1585.78} C_VEL
LIN {X 0,Y 587.358,Z 332.323,A -85,B 0,C 180,E1 -1588.232,E2 -1588.232} C_VEL
LIN {X 0,Y 587.354,Z 332.325,A -85,B 0,C 180,E1 -1590.867,E2 -1590.867} C_VEL
LIN {X 0,Y 587.342,Z 332.325,A -85,B 0,C 180,E1 -1593.722,E2 -1593.722} C_VEL
LIN {X 0,Y 587.344,Z 332.324,A -85,B 0,C 180,E1 -1595.994,E2 -1595.994} C_VEL
LIN {X 0,Y 587.33,Z 332.326,A -85,B 0,C 180,E1 -1598.226,E2 -1598.226} C_VEL
LIN {X 0,Y 587.349,Z 332.324,A -85,B 0,C 180,E1 -1601.151,E2 -1601.151} C_VEL
LIN {X 0,Y 587.333,Z 332.327,A -85,B 0,C 180,E1 -1604.025,E2 -1604.025} C_VEL
LIN {X 0,Y 587.366,Z 332.322,A -85,B 0,C 180,E1 -1606.155,E2 -1606.155} C_VEL
LIN {X 0,Y 587.343,Z 332.325,A -85,B 0,C 180,E1 -1608.963,E2 -1608.963} C_VEL
LIN {X 0,Y 587.372,Z 332.321,A -85,B 0,C 180,E1 -1611.745,E2 -1611.745} C_VEL
LIN {X 0,Y 587.362,Z 332.323,A -85,B 0,C 180,E1 -1614.507,E2 -1614.507} C_VEL
LIN {X 0,Y 587.377,Z 332.32,A -85,B 0,C 180,E1 -1617.257,E2 -1617.257} C_VEL
LIN {X 0,Y 587.389,Z 332.321,A -85,B 0,C 180,E1 -1620,E2 -1620} C_VEL
LIN {X 0,Y 587.379,Z 332.32,A -85,B 0,C 180,E1 -1622.743,E2 -1622.743} C_VEL
LIN {X 0,Y 587.359,Z 332.325,A -85,B 0,C 180,E1 -1625.493,E2 -1625.493} C_VEL
LIN {X 0,Y 587.375,Z 332.32,A -85,B 0,C 180,E1 -1628.255,E2 -1628.255} C_VEL
LIN {X 0,Y 587.355,Z 332.326,A -85,B 0,C 180,E1 -1631.134,E2 -1631.134} C_VEL
LIN {X 0,Y 587.371,Z 332.322,A -85,B 0,C 180,E1 -1634.26,E2 -1634.26} C_VEL
LIN {X 0,Y 587.365,Z 332.322,A -85,B 0,C 180,E1 -1637.406,E2 -1637.406} C_VEL
LIN {X 0,Y 587.328,Z 332.326,A -85,B 0,C 180,E1 -1638.314,E2 -1638.314} C_VEL
LIN {X 0,Y 586.674,Z 332.41,A -85,B 0,C 180,E1 -1638.886,E2 -1638.886} C_VEL
LIN {X 0,Y 583.844,Z 332.765,A -85,B 0,C 180,E1 -1639.814,E2 -1639.814} C_VEL
LIN {X 0,Y 581.436,Z 333.066,A -85,B 0,C 180,E1 -1640.561,E2 -1640.561} C_VEL
LIN {X 0,Y 580.384,Z 333.195,A -85,B 0,C 180,E1 -1641.137,E2 -1641.137} C_VEL
LIN {X 0,Y 580.289,Z 333.205,A -85,B 0,C 180,E1 -1641.332,E2 -1641.332} C_VEL
LIN {X 0,Y 580.308,Z 333.202,A -85,B 0,C 180,E1 -1644.316,E2 -1644.316} C_VEL
LIN {X 0,Y 580.285,Z 333.205,A -85,B 0,C 180,E1 -1646.623,E2 -1646.623} C_VEL
LIN {X 0,Y 580.303,Z 333.202,A -85,B 0,C 180,E1 -1649.309,E2 -1649.309} C_VEL
LIN {X 0,Y 580.306,Z 333.202,A -85,B 0,C 180,E1 -1652.2,E2 -1652.2} C_VEL
LIN {X 0,Y 580.298,Z 333.205,A -85,B 0,C 180,E1 -1654.696,E2 -1654.696} C_VEL
LIN {X 0,Y 580.305,Z 333.202,A -85,B 0,C 180,E1 -1657.268,E2 -1657.268} C_VEL
LIN {X 0,Y 580.305,Z 333.204,A -85,B 0,C 180,E1 -1660.271,E2 -1660.271} C_VEL
LIN {X 0,Y 580.283,Z 333.205,A -85,B 0,C 180,E1 -1662.706,E2 -1662.706} C_VEL
LIN {X 0,Y 580.279,Z 333.205,A -85,B 0,C 180,E1 -1665.609,E2 -1665.609} C_VEL
LIN {X 0,Y 580.322,Z 333.201,A -85,B 0,C 180,E1 -1668.234,E2 -1668.234} C_VEL
LIN {X 0,Y 580.28,Z 333.204,A -85,B 0,C 180,E1 -1670.965,E2 -1670.965} C_VEL
LIN {X 0,Y 580.256,Z 333.209,A -85,B 0,C 180,E1 -1673.595,E2 -1673.595} C_VEL
LIN {X 0,Y 580.323,Z 333.2,A -85,B 0,C 180,E1 -1676.145,E2 -1676.145} C_VEL
LIN {X 0,Y 580.281,Z 333.204,A -85,B 0,C 180,E1 -1678.614,E2 -1678.614} C_VEL
LIN {X 0,Y 580.299,Z 333.202,A -85,B 0,C 180,E1 -1681.024,E2 -1681.024} C_VEL
LIN {X 0,Y 580.299,Z 333.204,A -85,B 0,C 180,E1 -1683.666,E2 -1683.666} C_VEL
LIN {X 0,Y 580.308,Z 333.201,A -85,B 0,C 180,E1 -1685.684,E2 -1685.684} C_VEL
LIN {X 0,Y 580.276,Z 333.205,A -85,B 0,C 180,E1 -1687.947,E2 -1687.947} C_VEL
LIN {X 0,Y 580.306,Z 333.201,A -85,B 0,C 180,E1 -1690.913,E2 -1690.913} C_VEL
LIN {X 0,Y 580.284,Z 333.206,A -85,B 0,C 180,E1 -1693.825,E2 -1693.825} C_VEL
LIN {X 0,Y 580.332,Z 333.199,A -85,B 0,C 180,E1 -1695.983,E2 -1695.983} C_VEL
LIN {X 0,Y 580.313,Z 333.2,A -85,B 0,C 180,E1 -1698.827,E2 -1698.827} C_VEL
LIN {X 0,Y 580.335,Z 333.199,A -85,B 0,C 180,E1 -1701.644,E2 -1701.644} C_VEL
LIN {X 0,Y 580.324,Z 333.199,A -85,B 0,C 180,E1 -1704.44,E2 -1704.44} C_VEL
LIN {X 0,Y 580.299,Z 333.248,A -85,B 0,C 180,E1 -1705.919,E2 -1705.919} C_VEL
LIN {X 0,Y 580.743,Z 337.148,A -85,B 0,C 180,E1 -1706.031,E2 -1706.031} C_VEL
LIN {X 0,Y 580.657,Z 349.404,A -85,B 0,C 180,E1 -1706.443,E2 -1706.443} C_VEL
LIN {X 0,Y 580.562,Z 360.897,A -85,B 0,C 180,E1 -1706.964,E2 -1706.964} C_VEL
LIN {X 0,Y 580.508,Z 371.408,A -85,B 0,C 180,E1 -1707.571,E2 -1707.571} C_VEL
LIN {X 0,Y 580.402,Z 382.214,A -85,B 0,C 180,E1 -1708.352,E2 -1708.352} C_VEL
LIN {X 0,Y 580.273,Z 392.792,A -85,B 0,C 180,E1 -1709.306,E2 -1709.306} C_VEL
LIN {X 0,Y 580.221,Z 400.623,A -85,B 0,C 180,E1 -1710.173,E2 -1710.173} C_VEL
LIN {X 0,Y 580.171,Z 408.313,A -85,B 0,C 180,E1 -1711.214,E2 -1711.214} C_VEL
LIN {X 0,Y 580.112,Z 415.402,A -85,B 0,C 180,E1 -1712.43,E2 -1712.43} C_VEL
LIN {X 0,Y 580.127,Z 420.141,A -85,B 0,C 180,E1 -1713.472,E2 -1713.472} C_VEL
LIN {X 0,Y 580.104,Z 423.788,A -85,B 0,C 180,E1 -1714.516,E2 -1714.516} C_VEL
LIN {X 0,Y 580.099,Z 426.432,A -85,B 0,C 180,E1 -1715.561,E2 -1715.561} C_VEL
LIN {X 0,Y 580.101,Z 428.078,A -85,B 0,C 180,E1 -1716.561,E2 -1716.561} C_VEL
LIN {X 0,Y 580.067,Z 428.919,A -85,B 0,C 180,E1 -1717.658,E2 -1717.658} C_VEL
LIN {X 0,Y 580.061,Z 428.936,A -85,B 0,C 180,E1 -1718.359,E2 -1718.359} C_VEL
LIN {X 0,Y 580.026,Z 428.565,A -85,B 0,C 180,E1 -1719.062,E2 -1719.062} C_VEL
LIN {X 0,Y 580.058,Z 427.777,A -85,B 0,C 180,E1 -1719.765,E2 -1719.765} C_VEL
LIN {X 0,Y 580.074,Z 425.172,A -85,B 0,C 180,E1 -1721.074,E2 -1721.074} C_VEL
LIN {X 0,Y 580.081,Z 421.583,A -85,B 0,C 180,E1 -1722.24,E2 -1722.24} C_VEL
LIN {X 0,Y 580.097,Z 417.137,A -85,B 0,C 180,E1 -1723.308,E2 -1723.308} C_VEL
LIN {X 0,Y 580.156,Z 411.004,A -85,B 0,C 180,E1 -1724.453,E2 -1724.453} C_VEL
LIN {X 0,Y 580.199,Z 404.248,A -85,B 0,C 180,E1 -1725.455,E2 -1725.455} C_VEL
LIN {X 0,Y 580.263,Z 395.171,A -85,B 0,C 180,E1 -1726.536,E2 -1726.536} C_VEL
LIN {X 0,Y 580.359,Z 385.808,A -85,B 0,C 180,E1 -1727.44,E2 -1727.44} C_VEL
LIN {X 0,Y 580.446,Z 375.298,A -85,B 0,C 180,E1 -1728.257,E2 -1728.257} C_VEL
LIN {X 0,Y 580.567,Z 363.545,A -85,B 0,C 180,E1 -1728.985,E2 -1728.985} C_VEL
LIN {X 0,Y 580.661,Z 351.811,A -85,B 0,C 180,E1 -1729.551,E2 -1729.551} C_VEL
LIN {X 0,Y 580.741,Z 339.501,A -85,B 0,C 180,E1 -1729.991,E2 -1729.991} C_VEL
LIN {X 0,Y 580.483,Z 334.055,A -85,B 0,C 180,E1 -1730.147,E2 -1730.147} C_VEL
LIN {X 0,Y 580.312,Z 333.202,A -85,B 0,C 180,E1 -1730.191,E2 -1730.191} C_VEL
LIN {X 0,Y 580.274,Z 333.205,A -85,B 0,C 180,E1 -1733.003,E2 -1733.003} C_VEL
LIN {X 0,Y 580.31,Z 333.201,A -85,B 0,C 180,E1 -1735.079,E2 -1735.079} C_VEL
LIN {X 0,Y 580.299,Z 333.203,A -85,B 0,C 180,E1 -1738.185,E2 -1738.185} C_VEL
LIN {X 0,Y 580.285,Z 333.205,A -85,B 0,C 180,E1 -1740.694,E2 -1740.694} C_VEL
LIN {X 0,Y 580.307,Z 333.203,A -85,B 0,C 180,E1 -1743.316,E2 -1743.316} C_VEL
LIN {X 0,Y 580.249,Z 333.21,A -85,B 0,C 180,E1 -1745.756,E2 -1745.756} C_VEL
LIN {X 0,Y 580.289,Z 333.204,A -85,B 0,C 180,E1 -1748.146,E2 -1748.146} C_VEL
LIN {X 0,Y 580.301,Z 333.203,A -85,B 0,C 180,E1 -1750.843,E2 -1750.843} C_VEL
LIN {X 0,Y 580.289,Z 333.205,A -85,B 0,C 180,E1 -1753.656,E2 -1753.656} C_VEL
LIN {X 0,Y 580.277,Z 333.206,A -85,B 0,C 180,E1 -1756.609,E2 -1756.609} C_VEL
LIN {X 0,Y 580.302,Z 333.203,A -85,B 0,C 180,E1 -1759.156,E2 -1759.156} C_VEL
LIN {X 0,Y 580.291,Z 333.204,A -85,B 0,C 180,E1 -1761.926,E2 -1761.926} C_VEL
LIN {X 0,Y 580.309,Z 333.204,A -85,B 0,C 180,E1 -1764.456,E2 -1764.456} C_VEL
LIN {X 0,Y 580.292,Z 333.203,A -85,B 0,C 180,E1 -1766.975,E2 -1766.975} C_VEL
LIN {X 0,Y 580.31,Z 333.2,A -85,B 0,C 180,E1 -1769.426,E2 -1769.426} C_VEL
LIN {X 0,Y 580.32,Z 333.199,A -85,B 0,C 180,E1 -1772.136,E2 -1772.136} C_VEL
LIN {X 0,Y 580.309,Z 333.201,A -85,B 0,C 180,E1 -1774.92,E2 -1774.92} C_VEL
LIN {X 0,Y 580.276,Z 333.205,A -85,B 0,C 180,E1 -1777.947,E2 -1777.947} C_VEL
LIN {X 0,Y 580.317,Z 333.2,A -85,B 0,C 180,E1 -1780.914,E2 -1780.914} C_VEL
LIN {X 0,Y 580.284,Z 333.204,A -85,B 0,C 180,E1 -1783.825,E2 -1783.825} C_VEL
LIN {X 0,Y 580.281,Z 333.205,A -85,B 0,C 180,E1 -1786.696,E2 -1786.696} C_VEL
LIN {X 0,Y 580.303,Z 333.202,A -85,B 0,C 180,E1 -1789.533,E2 -1789.533} C_VEL
LIN {X 0,Y 580.328,Z 333.201,A -85,B 0,C 180,E1 -1792.344,E2 -1792.344} C_VEL
LIN {X 0,Y 580.34,Z 333.197,A -85,B 0,C 180,E1 -1795.137,E2 -1795.137} C_VEL
LIN {X 0,Y 580.335,Z 333.198,A -85,B 0,C 180,E1 -1797.918,E2 -1797.918} C_VEL
LIN {X 0,Y 580.365,Z 333.194,A -85,B 0,C 180,E1 -1800.694,E2 -1800.694} C_VEL
LIN {X 0,Y 580.287,Z 333.205,A -85,B 0,C 180,E1 -1803.472,E2 -1803.472} C_VEL
LIN {X 0,Y 580.327,Z 333.199,A -85,B 0,C 180,E1 -1805.56,E2 -1805.56} C_VEL
LIN {X 0,Y 580.331,Z 333.2,A -85,B 0,C 180,E1 -1808.356,E2 -1808.356} C_VEL
LIN {X 0,Y 580.296,Z 333.204,A -85,B 0,C 180,E1 -1811.191,E2 -1811.191} C_VEL
LIN {X 0,Y 580.324,Z 333.199,A -85,B 0,C 180,E1 -1814.017,E2 -1814.017} C_VEL
LIN {X 0,Y 580.309,Z 333.201,A -85,B 0,C 180,E1 -1816.914,E2 -1816.914} C_VEL
LIN {X 0,Y 580.303,Z 333.202,A -85,B 0,C 180,E1 -1819.822,E2 -1819.822} C_VEL
LIN {X 0,Y 580.293,Z 333.203,A -85,B 0,C 180,E1 -1822.803,E2 -1822.803} C_VEL
LIN {X 0,Y 580.305,Z 333.204,A -85,B 0,C 180,E1 -1825.08,E2 -1825.08} C_VEL
LIN {X 0,Y 580.317,Z 333.201,A -85,B 0,C 180,E1 -1827.863,E2 -1827.863} C_VEL
LIN {X 0,Y 580.298,Z 333.203,A -85,B 0,C 180,E1 -1830.698,E2 -1830.698} C_VEL
LIN {X 0,Y 580.303,Z 333.203,A -85,B 0,C 180,E1 -1833.317,E2 -1833.317} C_VEL
LIN {X 0,Y 580.325,Z 333.199,A -85,B 0,C 180,E1 -1835.768,E2 -1835.768} C_VEL
LIN {X 0,Y 580.29,Z 333.205,A -85,B 0,C 180,E1 -1838.146,E2 -1838.146} C_VEL
LIN {X 0,Y 580.319,Z 333.2,A -85,B 0,C 180,E1 -1840.842,E2 -1840.842} C_VEL
LIN {X 0,Y 580.287,Z 333.204,A -85,B 0,C 180,E1 -1843.657,E2 -1843.657} C_VEL
LIN {X 0,Y 580.292,Z 333.203,A -85,B 0,C 180,E1 -1846.608,E2 -1846.608} C_VEL
LIN {X 0,Y 580.321,Z 333.203,A -85,B 0,C 180,E1 -1849.159,E2 -1849.159} C_VEL
LIN {X 0,Y 580.292,Z 333.206,A -85,B 0,C 180,E1 -1851.927,E2 -1851.927} C_VEL
LIN {X 0,Y 580.373,Z 333.387,A -85,B 0,C 180,E1 -1853.692,E2 -1853.692} C_VEL
LIN {X 0,Y 580.919,Z 338.76,A -85,B 0,C 180,E1 -1854.925,E2 -1854.925} C_VEL
LIN {X 0,Y 580.711,Z 352.583,A -85,B 0,C 180,E1 -1857.905,E2 -1857.905} C_VEL
LIN {X 0,Y 580.754,Z 365.699,A -85,B 0,C 180,E1 -1860.611,E2 -1860.611} C_VEL
LIN {X 0,Y 580.802,Z 377.577,A -85,B 0,C 180,E1 -1863.015,E2 -1863.015} C_VEL
LIN {X 0,Y 580.666,Z 390.488,A -85,B 0,C 180,E1 -1865.701,E2 -1865.701} C_VEL
LIN {X 0,Y 580.563,Z 403.199,A -85,B 0,C 180,E1 -1868.333,E2 -1868.333} C_VEL
LIN {X 0,Y 580.42,Z 417.726,A -85,B 0,C 180,E1 -1871.285,E2 -1871.285} C_VEL
LIN {X 0,Y 580.324,Z 430.437,A -85,B 0,C 180,E1 -1873.827,E2 -1873.827} C_VEL
LIN {X 0,Y 580.287,Z 443.148,A -85,B 0,C 180,E1 -1876.34,E2 -1876.34} C_VEL
LIN {X 0,Y 580.271,Z 449.882,A -85,B 0,C 180,E1 -1877.619,E2 -1877.619} C_VEL
LIN {X 0,Y 580.816,Z 454.973,A -85,B 0,C 180,E1 -1877.709,E2 -1877.709} C_VEL
LIN {X 0,Y 580.724,Z 468.237,A -85,B 0,C 180,E1 -1878.017,E2 -1878.017} C_VEL
LIN {X 0,Y 580.657,Z 479.928,A -85,B 0,C 180,E1 -1878.419,E2 -1878.419} C_VEL
LIN {X 0,Y 580.567,Z 490.938,A -85,B 0,C 180,E1 -1878.921,E2 -1878.921} C_VEL
LIN {X 0,Y 580.477,Z 501.592,A -85,B 0,C 180,E1 -1879.537,E2 -1879.537} C_VEL
LIN {X 0,Y 580.38,Z 512.48,A -85,B 0,C 180,E1 -1880.328,E2 -1880.328} C_VEL
LIN {X 0,Y 580.271,Z 523.117,A -85,B 0,C 180,E1 -1881.293,E2 -1881.293} C_VEL
LIN {X 0,Y 580.221,Z 530.965,A -85,B 0,C 180,E1 -1882.169,E2 -1882.169} C_VEL
LIN {X 0,Y 580.153,Z 538.653,A -85,B 0,C 180,E1 -1883.222,E2 -1883.222} C_VEL
LIN {X 0,Y 580.139,Z 545.683,A -85,B 0,C 180,E1 -1884.439,E2 -1884.439} C_VEL
LIN {X 0,Y 580.108,Z 550.374,A -85,B 0,C 180,E1 -1885.484,E2 -1885.484} C_VEL
LIN {X 0,Y 580.123,Z 553.958,A -85,B 0,C 180,E1 -1886.528,E2 -1886.528} C_VEL
LIN {X 0,Y 580.043,Z 555.81,A -85,B 0,C 180,E1 -1887.223,E2 -1887.223} C_VEL
LIN {X 0,Y 580.04,Z 557.2,A -85,B 0,C 180,E1 -1887.917,E2 -1887.917} C_VEL
LIN {X 0,Y 580.04,Z 558.785,A -85,B 0,C 180,E1 -1889.306,E2 -1889.306} C_VEL
LIN {X 0,Y 580.037,Z 559,A -85,B 0,C 180,E1 -1890.001,E2 -1890.001} C_VEL
LIN {X 0,Y 580.047,Z 558.185,A -85,B 0,C 180,E1 -1891.389,E2 -1891.389} C_VEL
LIN {X 0,Y 580.04,Z 557.2,A -85,B 0,C 180,E1 -1892.084,E2 -1892.084} C_VEL
LIN {X 0,Y 580.043,Z 555.809,A -85,B 0,C 180,E1 -1892.778,E2 -1892.778} C_VEL
LIN {X 0,Y 580.109,Z 552.894,A -85,B 0,C 180,E1 -1893.821,E2 -1893.821} C_VEL
LIN {X 0,Y 580.054,Z 548.947,A -85,B 0,C 180,E1 -1894.866,E2 -1894.866} C_VEL
LIN {X 0,Y 580.139,Z 542.874,A -85,B 0,C 180,E1 -1896.085,E2 -1896.085} C_VEL
LIN {X 0,Y 580.185,Z 536.233,A -85,B 0,C 180,E1 -1897.133,E2 -1897.133} C_VEL
LIN {X 0,Y 580.251,Z 527.986,A -85,B 0,C 180,E1 -1898.182,E2 -1898.182} C_VEL
LIN {X 0,Y 580.308,Z 519.532,A -85,B 0,C 180,E1 -1899.059,E2 -1899.059} C_VEL
LIN {X 0,Y 580.425,Z 509.089,A -85,B 0,C 180,E1 -1899.936,E2 -1899.936} C_VEL
LIN {X 0,Y 580.492,Z 498.749,A -85,B 0,C 180,E1 -1900.64,E2 -1900.64} C_VEL
LIN {X 0,Y 580.597,Z 487.241,A -85,B 0,C 180,E1 -1901.264,E2 -1901.264} C_VEL
LIN {X 0,Y 580.691,Z 474.456,A -85,B 0,C 180,E1 -1901.785,E2 -1901.785} C_VEL
LIN {X 0,Y 580.775,Z 461.414,A -85,B 0,C 180,E1 -1902.16,E2 -1902.16} C_VEL
LIN {X 0,Y 580.611,Z 452.074,A -85,B 0,C 180,E1 -1902.341,E2 -1902.341} C_VEL
LIN {X 0,Y 580.244,Z 449.612,A -85,B 0,C 180,E1 -1902.393,E2 -1902.393} C_VEL
LIN {X 0,Y 580.325,Z 435.879,A -85,B 0,C 180,E1 -1905.093,E2 -1905.093} C_VEL
LIN {X 0,Y 580.389,Z 423.168,A -85,B 0,C 180,E1 -1907.622,E2 -1907.622} C_VEL
LIN {X 0,Y 580.471,Z 410.457,A -85,B 0,C 180,E1 -1910.186,E2 -1910.186} C_VEL
LIN {X 0,Y 580.606,Z 397.746,A -85,B 0,C 180,E1 -1912.79,E2 -1912.79} C_VEL
LIN {X 0,Y 580.751,Z 383.22,A -85,B 0,C 180,E1 -1915.828,E2 -1915.828} C_VEL
LIN {X 0,Y 580.763,Z 371.727,A -85,B 0,C 180,E1 -1918.162,E2 -1918.162} C_VEL
LIN {X 0,Y 580.769,Z 357.804,A -85,B 0,C 180,E1 -1921.024,E2 -1921.024} C_VEL
LIN {X 0,Y 580.833,Z 344.638,A -85,B 0,C 180,E1 -1923.821,E2 -1923.821} C_VEL
LIN {X 0,Y 580.886,Z 337.009,A -85,B 0,C 180,E1 -1925.503,E2 -1925.503} C_VEL
LIN {X 0,Y 580.279,Z 333.206,A -85,B 0,C 180,E1 -1926.403,E2 -1926.403} C_VEL
LIN {X 0,Y 580.296,Z 333.204,A -85,B 0,C 180,E1 -1929.185,E2 -1929.185} C_VEL
LIN {X 0,Y 580.319,Z 333.202,A -85,B 0,C 180,E1 -1931.766,E2 -1931.766} C_VEL
LIN {X 0,Y 580.275,Z 333.206,A -85,B 0,C 180,E1 -1934.626,E2 -1934.626} C_VEL
LIN {X 0,Y 580.29,Z 333.203,A -85,B 0,C 180,E1 -1937.628,E2 -1937.628} C_VEL
LIN {X 0,Y 580.3,Z 333.201,A -85,B 0,C 180,E1 -1940.068,E2 -1940.068} C_VEL
LIN {X 0,Y 580.304,Z 333.203,A -85,B 0,C 180,E1 -1943.066,E2 -1943.066} C_VEL
LIN {X 0,Y 580.321,Z 333.201,A -85,B 0,C 180,E1 -1946.146,E2 -1946.146} C_VEL
LIN {X 0,Y 580.294,Z 333.205,A -85,B 0,C 180,E1 -1948.616,E2 -1948.616} C_VEL
LIN {X 0,Y 580.296,Z 333.203,A -85,B 0,C 180,E1 -1951.024,E2 -1951.024} C_VEL
LIN {X 0,Y 580.295,Z 333.202,A -85,B 0,C 180,E1 -1953.667,E2 -1953.667} C_VEL
LIN {X 0,Y 580.307,Z 333.2,A -85,B 0,C 180,E1 -1955.684,E2 -1955.684} C_VEL
LIN {X 0,Y 580.28,Z 333.204,A -85,B 0,C 180,E1 -1957.948,E2 -1957.948} C_VEL
LIN {X 0,Y 580.301,Z 333.204,A -85,B 0,C 180,E1 -1960.914,E2 -1960.914} C_VEL
LIN {X 0,Y 580.286,Z 333.203,A -85,B 0,C 180,E1 -1963.826,E2 -1963.826} C_VEL
LIN {X 0,Y 580.332,Z 333.198,A -85,B 0,C 180,E1 -1965.983,E2 -1965.983} C_VEL
LIN {X 0,Y 580.311,Z 333.202,A -85,B 0,C 180,E1 -1968.827,E2 -1968.827} C_VEL
LIN {X 0,Y 580.335,Z 333.197,A -85,B 0,C 180,E1 -1971.644,E2 -1971.644} C_VEL
LIN {X 0,Y 580.328,Z 333.2,A -85,B 0,C 180,E1 -1974.44,E2 -1974.44} C_VEL
LIN {X 0,Y 580.344,Z 333.196,A -85,B 0,C 180,E1 -1977.224,E2 -1977.224} C_VEL
LIN {X 0,Y 580.359,Z 333.197,A -85,B 0,C 180,E1 -1980,E2 -1980} C_VEL
LIN {X 0,Y 580.345,Z 333.196,A -85,B 0,C 180,E1 -1982.777,E2 -1982.777} C_VEL
LIN {X 0,Y 580.325,Z 333.201,A -85,B 0,C 180,E1 -1985.56,E2 -1985.56} C_VEL
LIN {X 0,Y 580.34,Z 333.197,A -85,B 0,C 180,E1 -1988.356,E2 -1988.356} C_VEL
LIN {X 0,Y 580.307,Z 333.203,A -85,B 0,C 180,E1 -1991.191,E2 -1991.191} C_VEL
LIN {X 0,Y 580.331,Z 333.198,A -85,B 0,C 180,E1 -1994.017,E2 -1994.017} C_VEL
LIN {X 0,Y 580.319,Z 333.201,A -85,B 0,C 180,E1 -1996.914,E2 -1996.914} C_VEL
LIN {X 0,Y 580.292,Z 333.204,A -85,B 0,C 180,E1 -1999.823,E2 -1999.823} C_VEL
LIN {X 0,Y 580.289,Z 333.205,A -85,B 0,C 180,E1 -2001.332,E2 -2001.332} C_VEL
LIN {X 0,Y 579.592,Z 333.291,A -85,B 0,C 180,E1 -2001.912,E2 -2001.912} C_VEL
LIN {X 0,Y 576.715,Z 333.648,A -85,B 0,C 180,E1 -2002.852,E2 -2002.852} C_VEL
LIN {X 0,Y 574.322,Z 333.948,A -85,B 0,C 180,E1 -2003.608,E2 -2003.608} C_VEL
LIN {X 0,Y 573.324,Z 334.071,A -85,B 0,C 180,E1 -2004.192,E2 -2004.192} C_VEL
LIN {X 0,Y 573.257,Z 334.079,A -85,B 0,C 180,E1 -2004.389,E2 -2004.389} C_VEL
LIN {X 0,Y 573.258,Z 334.081,A -85,B 0,C 180,E1 -2006.976,E2 -2006.976} C_VEL
LIN {X 0,Y 573.249,Z 334.08,A -85,B 0,C 180,E1 -2009.487,E2 -2009.487} C_VEL
LIN {X 0,Y 573.262,Z 334.079,A -85,B 0,C 180,E1 -2012.645,E2 -2012.645} C_VEL
LIN {X 0,Y 573.216,Z 334.084,A -85,B 0,C 180,E1 -2015.188,E2 -2015.188} C_VEL
LIN {X 0,Y 573.243,Z 334.082,A -85,B 0,C 180,E1 -2017.807,E2 -2017.807} C_VEL
LIN {X 0,Y 573.277,Z 334.077,A -85,B 0,C 180,E1 -2020.528,E2 -2020.528} C_VEL
LIN {X 0,Y 573.245,Z 334.083,A -85,B 0,C 180,E1 -2023.668,E2 -2023.668} C_VEL
LIN {X 0,Y 573.255,Z 334.079,A -85,B 0,C 180,E1 -2026.642,E2 -2026.642} C_VEL
LIN {X 0,Y 573.252,Z 334.081,A -85,B 0,C 180,E1 -2029.475,E2 -2029.475} C_VEL
LIN {X 0,Y 573.237,Z 334.081,A -85,B 0,C 180,E1 -2032.192,E2 -2032.192} C_VEL
LIN {X 0,Y 573.242,Z 334.081,A -85,B 0,C 180,E1 -2035.229,E2 -2035.229} C_VEL
LIN {X 0,Y 573.259,Z 334.079,A -85,B 0,C 180,E1 -2037.772,E2 -2037.772} C_VEL
LIN {X 0,Y 573.266,Z 334.08,A -85,B 0,C 180,E1 -2040.634,E2 -2040.634} C_VEL
LIN {X 0,Y 573.244,Z 334.081,A -85,B 0,C 180,E1 -2043.507,E2 -2043.507} C_VEL
LIN {X 0,Y 573.239,Z 334.084,A -85,B 0,C 180,E1 -2046.134,E2 -2046.134} C_VEL
LIN {X 0,Y 573.258,Z 334.08,A -85,B 0,C 180,E1 -2049.173,E2 -2049.173} C_VEL
LIN {X 0,Y 573.23,Z 334.083,A -85,B 0,C 180,E1 -2051.411,E2 -2051.411} C_VEL
LIN {X 0,Y 573.256,Z 334.08,A -85,B 0,C 180,E1 -2053.621,E2 -2053.621} C_VEL
LIN {X 0,Y 573.28,Z 334.076,A -85,B 0,C 180,E1 -2055.807,E2 -2055.807} C_VEL
LIN {X 0,Y 573.271,Z 334.078,A -85,B 0,C 180,E1 -2058.745,E2 -2058.745} C_VEL
LIN {X 0,Y 573.291,Z 334.076,A -85,B 0,C 180,E1 -2061.54,E2 -2061.54} C_VEL
LIN {X 0,Y 573.291,Z 334.076,A -85,B 0,C 180,E1 -2064.371,E2 -2064.371} C_VEL
LIN {X 0,Y 573.232,Z 334.083,A -85,B 0,C 180,E1 -2065.781,E2 -2065.781} C_VEL
LIN {X 0,Y 573.79,Z 337.543,A -85,B 0,C 180,E1 -2065.895,E2 -2065.895} C_VEL
LIN {X 0,Y 573.694,Z 350.798,A -85,B 0,C 180,E1 -2066.356,E2 -2066.356} C_VEL
LIN {X 0,Y 573.565,Z 362.783,A -85,B 0,C 180,E1 -2066.927,E2 -2066.927} C_VEL
LIN {X 0,Y 573.435,Z 374.184,A -85,B 0,C 180,E1 -2067.629,E2 -2067.629} C_VEL
LIN {X 0,Y 573.324,Z 384.464,A -85,B 0,C 180,E1 -2068.419,E2 -2068.419} C_VEL
LIN {X 0,Y 573.224,Z 393.775,A -85,B 0,C 180,E1 -2069.297,E2 -2069.297} C_VEL
LIN {X 0,Y 573.141,Z 402.777,A -85,B 0,C 180,E1 -2070.351,E2 -2070.351} C_VEL
LIN {X 0,Y 573.039,Z 410.06,A -85,B 0,C 180,E1 -2071.405,E2 -2071.405} C_VEL
LIN {X 0,Y 573.033,Z 415.912,A -85,B 0,C 180,E1 -2072.46,E2 -2072.46} C_VEL
LIN {X 0,Y 573.054,Z 420.542,A -85,B 0,C 180,E1 -2073.515,E2 -2073.515} C_VEL
LIN {X 0,Y 573.005,Z 424.088,A -85,B 0,C 180,E1 -2074.572,E2 -2074.572} C_VEL
LIN {X 0,Y 573,Z 426.635,A -85,B 0,C 180,E1 -2075.631,E2 -2075.631} C_VEL
LIN {X 0,Y 573.012,Z 428.084,A -85,B 0,C 180,E1 -2076.549,E2 -2076.549} C_VEL
LIN {X 0,Y 572.978,Z 428.942,A -85,B 0,C 180,E1 -2077.754,E2 -2077.754} C_VEL
LIN {X 0,Y 572.951,Z 428.913,A -85,B 0,C 180,E1 -2078.464,E2 -2078.464} C_VEL
LIN {X 0,Y 572.926,Z 428.487,A -85,B 0,C 180,E1 -2079.176,E2 -2079.176} C_VEL
LIN {X 0,Y 572.975,Z 427.619,A -85,B 0,C 180,E1 -2079.887,E2 -2079.887} C_VEL
LIN {X 0,Y 572.987,Z 425.171,A -85,B 0,C 180,E1 -2081.112,E2 -2081.112} C_VEL
LIN {X 0,Y 573.011,Z 421.225,A -85,B 0,C 180,E1 -2082.394,E2 -2082.394} C_VEL
LIN {X 0,Y 573.031,Z 416.67,A -85,B 0,C 180,E1 -2083.475,E2 -2083.475} C_VEL
LIN {X 0,Y 573.095,Z 409.756,A -85,B 0,C 180,E1 -2084.733,E2 -2084.733} C_VEL
LIN {X 0,Y 573.153,Z 402.063,A -85,B 0,C 180,E1 -2085.832,E2 -2085.832} C_VEL
LIN {X 0,Y 573.217,Z 394.666,A -85,B 0,C 180,E1 -2086.696,E2 -2086.696} C_VEL
LIN {X 0,Y 573.38,Z 384.594,A -85,B 0,C 180,E1 -2087.659,E2 -2087.659} C_VEL
LIN {X 0,Y 573.446,Z 373.791,A -85,B 0,C 180,E1 -2088.488,E2 -2088.488} C_VEL
LIN {X 0,Y 573.602,Z 362.171,A -85,B 0,C 180,E1 -2089.197,E2 -2089.197} C_VEL
LIN {X 0,Y 573.67,Z 349.65,A -85,B 0,C 180,E1 -2089.781,E2 -2089.781} C_VEL
LIN {X 0,Y 573.827,Z 336.325,A -85,B 0,C 180,E1 -2090.23,E2 -2090.23} C_VEL
LIN {X 0,Y 573.267,Z 334.08,A -85,B 0,C 180,E1 -2090.309,E2 -2090.309} C_VEL
LIN {X 0,Y 573.226,Z 334.083,A -85,B 0,C 180,E1 -2093.141,E2 -2093.141} C_VEL
LIN {X 0,Y 573.258,Z 334.081,A -85,B 0,C 180,E1 -2095.409,E2 -2095.409} C_VEL
LIN {X 0,Y 573.239,Z 334.084,A -85,B 0,C 180,E1 -2098.564,E2 -2098.564} C_VEL
LIN {X 0,Y 573.227,Z 334.083,A -85,B 0,C 180,E1 -2100.993,E2 -2100.993} C_VEL
LIN {X 0,Y 573.264,Z 334.081,A -85,B 0,C 180,E1 -2103.523,E2 -2103.523} C_VEL
LIN {X 0,Y 573.216,Z 334.085,A -85,B 0,C 180,E1 -2106.051,E2 -2106.051} C_VEL
LIN {X 0,Y 573.244,Z 334.082,A -85,B 0,C 180,E1 -2108.701,E2 -2108.701} C_VEL
LIN {X 0,Y 573.255,Z 334.081,A -85,B 0,C 180,E1 -2111.595,E2 -2111.595} C_VEL
LIN {X 0,Y 573.24,Z 334.083,A -85,B 0,C 180,E1 -2114.332,E2 -2114.332} C_VEL
LIN {X 0,Y 573.241,Z 334.083,A -85,B 0,C 180,E1 -2117.358,E2 -2117.358} C_VEL
LIN {X 0,Y 573.249,Z 334.082,A -85,B 0,C 180,E1 -2120.393,E2 -2120.393} C_VEL
LIN {X 0,Y 573.257,Z 334.08,A -85,B 0,C 180,E1 -2123.077,E2 -2123.077} C_VEL
LIN {X 0,Y 573.276,Z 334.078,A -85,B 0,C 180,E1 -2125.671,E2 -2125.671} C_VEL
LIN {X 0,Y 573.25,Z 334.08,A -85,B 0,C 180,E1 -2128.185,E2 -2128.185} C_VEL
LIN {X 0,Y 573.27,Z 334.076,A -85,B 0,C 180,E1 -2130.634,E2 -2130.634} C_VEL
LIN {X 0,Y 573.272,Z 334.079,A -85,B 0,C 180,E1 -2133.499,E2 -2133.499} C_VEL
LIN {X 0,Y 573.234,Z 334.082,A -85,B 0,C 180,E1 -2136.134,E2 -2136.134} C_VEL
LIN {X 0,Y 573.261,Z 334.08,A -85,B 0,C 180,E1 -2139.174,E2 -2139.174} C_VEL
LIN {X 0,Y 573.239,Z 334.083,A -85,B 0,C 180,E1 -2141.412,E2 -2141.412} C_VEL
LIN {X 0,Y 573.26,Z 334.08,A -85,B 0,C 180,E1 -2143.622,E2 -2143.622} C_VEL
LIN {X 0,Y 573.239,Z 334.083,A -85,B 0,C 180,E1 -2146.529,E2 -2146.529} C_VEL
LIN {X 0,Y 573.282,Z 334.077,A -85,B 0,C 180,E1 -2148.734,E2 -2148.734} C_VEL
LIN {X 0,Y 573.307,Z 334.074,A -85,B 0,C 180,E1 -2151.541,E2 -2151.541} C_VEL
LIN {X 0,Y 573.291,Z 334.076,A -85,B 0,C 180,E1 -2154.372,E2 -2154.372} C_VEL
LIN {X 0,Y 573.306,Z 334.073,A -85,B 0,C 180,E1 -2157.892,E2 -2157.892} C_VEL
LIN {X 0,Y 573.335,Z 334.069,A -85,B 0,C 180,E1 -2160.702,E2 -2160.702} C_VEL
LIN {X 0,Y 573.239,Z 334.082,A -85,B 0,C 180,E1 -2163.514,E2 -2163.514} C_VEL
LIN {X 0,Y 573.293,Z 334.075,A -85,B 0,C 180,E1 -2165.628,E2 -2165.628} C_VEL
LIN {X 0,Y 573.288,Z 334.076,A -85,B 0,C 180,E1 -2168.459,E2 -2168.459} C_VEL
LIN {X 0,Y 573.268,Z 334.08,A -85,B 0,C 180,E1 -2171.312,E2 -2171.312} C_VEL
LIN {X 0,Y 573.271,Z 334.079,A -85,B 0,C 180,E1 -2174.193,E2 -2174.193} C_VEL
LIN {X 0,Y 573.257,Z 334.081,A -85,B 0,C 180,E1 -2177.112,E2 -2177.112} C_VEL
LIN {X 0,Y 573.25,Z 334.082,A -85,B 0,C 180,E1 -2180.077,E2 -2180.077} C_VEL
LIN {X 0,Y 573.231,Z 334.085,A -85,B 0,C 180,E1 -2183.1,E2 -2183.1} C_VEL
LIN {X 0,Y 573.253,Z 334.081,A -85,B 0,C 180,E1 -2185.41,E2 -2185.41} C_VEL
LIN {X 0,Y 573.261,Z 334.081,A -85,B 0,C 180,E1 -2188.032,E2 -2188.032} C_VEL
LIN {X 0,Y 573.243,Z 334.082,A -85,B 0,C 180,E1 -2190.885,E2 -2190.885} C_VEL
LIN {X 0,Y 573.286,Z 334.076,A -85,B 0,C 180,E1 -2193.528,E2 -2193.528} C_VEL
LIN {X 0,Y 573.259,Z 334.081,A -85,B 0,C 180,E1 -2196.048,E2 -2196.048} C_VEL
LIN {X 0,Y 573.251,Z 334.079,A -85,B 0,C 180,E1 -2198.701,E2 -2198.701} C_VEL
LIN {X 0,Y 573.264,Z 334.077,A -85,B 0,C 180,E1 -2201.598,E2 -2201.598} C_VEL
LIN {X 0,Y 573.238,Z 334.082,A -85,B 0,C 180,E1 -2204.333,E2 -2204.333} C_VEL
LIN {X 0,Y 573.26,Z 334.08,A -85,B 0,C 180,E1 -2207.357,E2 -2207.357} C_VEL
LIN {X 0,Y 573.251,Z 334.082,A -85,B 0,C 180,E1 -2210.394,E2 -2210.394} C_VEL
LIN {X 0,Y 573.319,Z 334.192,A -85,B 0,C 180,E1 -2213.467,E2 -2213.467} C_VEL
LIN {X 0,Y 573.959,Z 338.248,A -85,B 0,C 180,E1 -2214.436,E2 -2214.436} C_VEL
LIN {X 0,Y 573.777,Z 349.751,A -85,B 0,C 180,E1 -2216.972,E2 -2216.972} C_VEL
LIN {X 0,Y 573.78,Z 363.335,A -85,B 0,C 180,E1 -2219.855,E2 -2219.855} C_VEL
LIN {X 0,Y 573.751,Z 376.898,A -85,B 0,C 180,E1 -2222.656,E2 -2222.656} C_VEL
LIN {X 0,Y 573.7,Z 390.488,A -85,B 0,C 180,E1 -2225.386,E2 -2225.386} C_VEL
LIN {X 0,Y 573.595,Z 403.199,A -85,B 0,C 180,E1 -2228.056,E2 -2228.056} C_VEL
LIN {X 0,Y 573.433,Z 417.743,A -85,B 0,C 180,E1 -2231.051,E2 -2231.051} C_VEL
LIN {X 0,Y 573.314,Z 430.437,A -85,B 0,C 180,E1 -2233.624,E2 -2233.624} C_VEL
LIN {X 0,Y 573.214,Z 444.964,A -85,B 0,C 180,E1 -2236.53,E2 -2236.53} C_VEL
LIN {X 0,Y 573.225,Z 449.882,A -85,B 0,C 180,E1 -2237.465,E2 -2237.465} C_VEL
LIN {X 0,Y 573.875,Z 456.115,A -85,B 0,C 180,E1 -2237.58,E2 -2237.58} C_VEL
LIN {X 0,Y 573.777,Z 469.757,A -85,B 0,C 180,E1 -2237.915,E2 -2237.915} C_VEL
LIN {X 0,Y 573.692,Z 481.507,A -85,B 0,C 180,E1 -2238.339,E2 -2238.339} C_VEL
LIN {X 0,Y 573.607,Z 492.638,A -85,B 0,C 180,E1 -2238.874,E2 -2238.874} C_VEL
LIN {X 0,Y 573.432,Z 504.21,A -85,B 0,C 180,E1 -2239.586,E2 -2239.586} C_VEL
LIN {X 0,Y 573.334,Z 514.606,A -85,B 0,C 180,E1 -2240.386,E2 -2240.386} C_VEL
LIN {X 0,Y 573.24,Z 523.118,A -85,B 0,C 180,E1 -2241.185,E2 -2241.185} C_VEL
LIN {X 0,Y 573.16,Z 530.965,A -85,B 0,C 180,E1 -2242.072,E2 -2242.072} C_VEL
LIN {X 0,Y 573.073,Z 538.583,A -85,B 0,C 180,E1 -2243.127,E2 -2243.127} C_VEL
LIN {X 0,Y 573.07,Z 545.683,A -85,B 0,C 180,E1 -2244.37,E2 -2244.37} C_VEL
LIN {X 0,Y 573.028,Z 550.374,A -85,B 0,C 180,E1 -2245.428,E2 -2245.428} C_VEL
LIN {X 0,Y 573.022,Z 553.959,A -85,B 0,C 180,E1 -2246.485,E2 -2246.485} C_VEL
LIN {X 0,Y 572.959,Z 555.81,A -85,B 0,C 180,E1 -2247.188,E2 -2247.188} C_VEL
LIN {X 0,Y 572.939,Z 557.2,A -85,B 0,C 180,E1 -2247.892,E2 -2247.892} C_VEL
LIN {X 0,Y 572.941,Z 558.785,A -85,B 0,C 180,E1 -2249.298,E2 -2249.298} C_VEL
LIN {X 0,Y 572.938,Z 559,A -85,B 0,C 180,E1 -2250.001,E2 -2250.001} C_VEL
LIN {X 0,Y 572.946,Z 558.185,A -85,B 0,C 180,E1 -2251.406,E2 -2251.406} C_VEL
LIN {X 0,Y 572.94,Z 557.199,A -85,B 0,C 180,E1 -2252.109,E2 -2252.109} C_VEL
LIN {X 0,Y 572.959,Z 555.809,A -85,B 0,C 180,E1 -2252.813,E2 -2252.813} C_VEL
LIN {X 0,Y 573.014,Z 552.894,A -85,B 0,C 180,E1 -2253.868,E2 -2253.868} C_VEL
LIN {X 0,Y 572.963,Z 548.947,A -85,B 0,C 180,E1 -2254.926,E2 -2254.926} C_VEL
LIN {X 0,Y 573.065,Z 542.874,A -85,B 0,C 180,E1 -2256.161,E2 -2256.161} C_VEL
LIN {X 0,Y 573.12,Z 536.234,A -85,B 0,C 180,E1 -2257.221,E2 -2257.221} C_VEL
LIN {X 0,Y 573.201,Z 527.986,A -85,B 0,C 180,E1 -2258.284,E2 -2258.284} C_VEL
LIN {X 0,Y 573.287,Z 519.533,A -85,B 0,C 180,E1 -2259.171,E2 -2259.171} C_VEL
LIN {X 0,Y 573.429,Z 509.091,A -85,B 0,C 180,E1 -2260.059,E2 -2260.059} C_VEL
LIN {X 0,Y 573.546,Z 497.427,A -85,B 0,C 180,E1 -2260.853,E2 -2260.853} C_VEL
LIN {X 0,Y 573.652,Z 486.295,A -85,B 0,C 180,E1 -2261.447,E2 -2261.447} C_VEL
LIN {X 0,Y 573.745,Z 473.158,A -85,B 0,C 180,E1 -2261.975,E2 -2261.975} C_VEL
LIN {X 0,Y 573.853,Z 460.498,A -85,B 0,C 180,E1 -2262.331,E2 -2262.331} C_VEL
LIN {X 0,Y 573.795,Z 453.576,A -85,B 0,C 180,E1 -2262.467,E2 -2262.467} C_VEL
LIN {X 0,Y 573.185,Z 449.612,A -85,B 0,C 180,E1 -2262.548,E2 -2262.548} C_VEL
LIN {X 0,Y 573.295,Z 435.879,A -85,B 0,C 180,E1 -2265.282,E2 -2265.282} C_VEL
LIN {X 0,Y 573.383,Z 423.168,A -85,B 0,C 180,E1 -2267.845,E2 -2267.845} C_VEL
LIN {X 0,Y 573.477,Z 410.457,A -85,B 0,C 180,E1 -2270.443,E2 -2270.443} C_VEL
LIN {X 0,Y 573.652,Z 397.746,A -85,B 0,C 180,E1 -2273.082,E2 -2273.082} C_VEL
LIN {X 0,Y 573.741,Z 384.77,A -85,B 0,C 180,E1 -2275.777,E2 -2275.777} C_VEL
LIN {X 0,Y 573.777,Z 373.114,A -85,B 0,C 180,E1 -2278.127,E2 -2278.127} C_VEL
LIN {X 0,Y 573.789,Z 359.481,A -85,B 0,C 180,E1 -2280.975,E2 -2280.975} C_VEL
LIN {X 0,Y 573.885,Z 345.832,A -85,B 0,C 180,E1 -2283.911,E2 -2283.911} C_VEL
LIN {X 0,Y 573.967,Z 338.434,A -85,B 0,C 180,E1 -2285.565,E2 -2285.565} C_VEL
LIN {X 0,Y 573.244,Z 334.082,A -85,B 0,C 180,E1 -2286.649,E2 -2286.649} C_VEL
LIN {X 0,Y 573.242,Z 334.083,A -85,B 0,C 180,E1 -2289.608,E2 -2289.608} C_VEL
LIN {X 0,Y 573.249,Z 334.082,A -85,B 0,C 180,E1 -2292.642,E2 -2292.642} C_VEL
LIN {X 0,Y 573.24,Z 334.081,A -85,B 0,C 180,E1 -2295.667,E2 -2295.667} C_VEL
LIN {X 0,Y 573.234,Z 334.084,A -85,B 0,C 180,E1 -2298.543,E2 -2298.543} C_VEL
LIN {X 0,Y 573.255,Z 334.079,A -85,B 0,C 180,E1 -2301.299,E2 -2301.299} C_VEL
LIN {X 0,Y 573.218,Z 334.086,A -85,B 0,C 180,E1 -2304.019,E2 -2304.019} C_VEL
LIN {X 0,Y 573.274,Z 334.078,A -85,B 0,C 180,E1 -2306.518,E2 -2306.518} C_VEL
LIN {X 0,Y 573.244,Z 334.081,A -85,B 0,C 180,E1 -2309.116,E2 -2309.116} C_VEL
LIN {X 0,Y 573.255,Z 334.081,A -85,B 0,C 180,E1 -2311.972,E2 -2311.972} C_VEL
LIN {X 0,Y 573.255,Z 334.08,A -85,B 0,C 180,E1 -2314.59,E2 -2314.59} C_VEL
LIN {X 0,Y 573.244,Z 334.082,A -85,B 0,C 180,E1 -2317.663,E2 -2317.663} C_VEL
LIN {X 0,Y 573.272,Z 334.079,A -85,B 0,C 180,E1 -2320.67,E2 -2320.67} C_VEL
LIN {X 0,Y 573.258,Z 334.078,A -85,B 0,C 180,E1 -2323.622,E2 -2323.622} C_VEL
LIN {X 0,Y 573.28,Z 334.076,A -85,B 0,C 180,E1 -2325.807,E2 -2325.807} C_VEL
LIN {X 0,Y 573.269,Z 334.08,A -85,B 0,C 180,E1 -2328.745,E2 -2328.745} C_VEL
LIN {X 0,Y 573.291,Z 334.074,A -85,B 0,C 180,E1 -2331.541,E2 -2331.541} C_VEL
LIN {X 0,Y 573.296,Z 334.077,A -85,B 0,C 180,E1 -2334.372,E2 -2334.372} C_VEL
LIN {X 0,Y 573.308,Z 334.074,A -85,B 0,C 180,E1 -2337.893,E2 -2337.893} C_VEL
LIN {X 0,Y 573.34,Z 334.069,A -85,B 0,C 180,E1 -2340.703,E2 -2340.703} C_VEL
LIN {X 0,Y 573.239,Z 334.082,A -85,B 0,C 180,E1 -2343.515,E2 -2343.515} C_VEL
LIN {X 0,Y 573.292,Z 334.077,A -85,B 0,C 180,E1 -2345.628,E2 -2345.628} C_VEL
LIN {X 0,Y 573.296,Z 334.074,A -85,B 0,C 180,E1 -2348.46,E2 -2348.46} C_VEL
LIN {X 0,Y 573.279,Z 334.078,A -85,B 0,C 180,E1 -2351.312,E2 -2351.312} C_VEL
LIN {X 0,Y 573.288,Z 334.078,A -85,B 0,C 180,E1 -2354.424,E2 -2354.424} C_VEL
LIN {X 0,Y 573.267,Z 334.078,A -85,B 0,C 180,E1 -2357.112,E2 -2357.112} C_VEL
LIN {X 0,Y 573.247,Z 334.083,A -85,B 0,C 180,E1 -2360.077,E2 -2360.077} C_VEL
LIN {X 0,Y 573.242,Z 334.083,A -85,B 0,C 180,E1 -2362.338,E2 -2362.338} C_VEL
LIN {X 0,Y 573.257,Z 334.079,A -85,B 0,C 180,E1 -2364.389,E2 -2364.389} C_VEL
